(* IEC 61131-3 sources: plc_simulator/services/codesys/POUs (part 5) *)

(* ---- STC_SortTasks.st ---- *)
(* ===========================================================================================
 *  STC_SortTasks — Insertion sort task queues by priority
 *
 *  Company : Galvatek part of the John Cockerill Group
 *  Author  : Jarmo Piipponen
 *  Created : 25.03.2026
 *
 * -------------------------------------------------------------------------------------------
 *  Shared FC: both TSK and DEP call this with different arrays.
 *  Priority: emergency (overtime ratio > 1.0) first, then
 *  earliest StartTime.
 *
 *  ------------------------------------------------------------------------------------------
 *
 *  Changes:
 *
 *
 *
 *)

FUNCTION STC_SortTasks : BOOL

(* Introduction of Variables ----------------------------------------------------------------*)

VAR_INPUT
  i_trans                   : INT;    (* 0 = all, 1..3 = specific transporter *)
  i_time_s                  : LINT;
END_VAR

VAR_IN_OUT  (* array sizes must match GVL_JC_Constants: 3=MAX_TRANSPORTERS, 10=MAX_UNITS *)
  io_task                   : ARRAY[1..3] OF UDT_JC_TskQueueType;
  io_batch                  : ARRAY[1..10] OF UDT_BatchType;
END_VAR

VAR_EXTERNAL CONSTANT
    MAX_TRANSPORTERS        : INT;
    MAX_UNITS               : INT;
    IN_PROCESS              : INT;
END_VAR

VAR_EXTERNAL
  g_unit                    : ARRAY[1..MAX_UNITS] OF UDT_JC_UnitType;
END_VAR

VAR
  ti                        : INT;
  t_start                   : INT;
  t_end                     : INT;
  ins_i                     : INT;
  ins_j                     : INT;
  ins_cnt                   : INT;
  tmp_task                  : UDT_JC_TskTaskType;
  tmp_unit                  : INT;
  cur_unit                  : INT;
  tmp_ratio                 : REAL;
  cur_ratio                 : REAL;
  tmp_emerg                 : BOOL;
  cur_emerg                 : BOOL;
  do_shift                  : BOOL;
END_VAR

STC_SortTasks := TRUE;

IF i_trans >= 1 AND i_trans <= 3 THEN
  t_start := i_trans;
  t_end   := i_trans;
ELSE
  t_start := 1;
  t_end   := 3;
END_IF;

FOR ti := t_start TO t_end DO
  ins_cnt := io_task[ti].Count;
  IF ins_cnt >= 2 THEN
    FOR ins_i := 2 TO ins_cnt DO
      tmp_task := io_task[ti].Queue[ins_i];

      tmp_ratio := 0.0;
      tmp_unit  := tmp_task.Unit;
      IF tmp_unit >= 1 AND tmp_unit <= MAX_UNITS THEN
        IF io_batch[tmp_unit].State = IN_PROCESS
           AND tmp_task.Stage >= 1 THEN
          IF io_batch[tmp_unit].CurStage = tmp_task.Stage
             AND g_unit[tmp_unit].location = tmp_task.LiftStationTarget
             AND io_batch[tmp_unit].StartTime > LINT#0
             AND io_batch[tmp_unit].MaxTime > 0 THEN
            tmp_ratio := LINT_TO_REAL(i_time_s - io_batch[tmp_unit].StartTime)
                         / DINT_TO_REAL(io_batch[tmp_unit].MaxTime);
          END_IF;
        END_IF;
      END_IF;
      tmp_emerg := tmp_ratio > 1.0;

      ins_j := 0;
      FOR ins_j := ins_i - 1 TO 1 BY -1 DO
        cur_ratio := 0.0;
        cur_unit  := io_task[ti].Queue[ins_j].Unit;
        IF cur_unit >= 1 AND cur_unit <= MAX_UNITS THEN
          IF io_batch[cur_unit].State = IN_PROCESS
             AND io_task[ti].Queue[ins_j].Stage >= 1 THEN
            IF io_batch[cur_unit].CurStage = io_task[ti].Queue[ins_j].Stage
               AND g_unit[cur_unit].location = io_task[ti].Queue[ins_j].LiftStationTarget
               AND io_batch[cur_unit].StartTime > LINT#0
               AND io_batch[cur_unit].MaxTime > 0 THEN
              cur_ratio := LINT_TO_REAL(i_time_s - io_batch[cur_unit].StartTime)
                           / DINT_TO_REAL(io_batch[cur_unit].MaxTime);
            END_IF;
          END_IF;
        END_IF;
        cur_emerg := cur_ratio > 1.0;

        do_shift := FALSE;
        IF tmp_emerg AND NOT cur_emerg THEN
          do_shift := TRUE;
        ELSIF tmp_emerg AND cur_emerg THEN
          IF tmp_ratio > cur_ratio THEN
            do_shift := TRUE;
          END_IF;
        ELSIF NOT tmp_emerg AND NOT cur_emerg THEN
          IF io_task[ti].Queue[ins_j].StartTime > tmp_task.StartTime THEN
            do_shift := TRUE;
          END_IF;
        END_IF;

        IF NOT do_shift THEN EXIT; END_IF;

        io_task[ti].Queue[ins_j + 1] := io_task[ti].Queue[ins_j];
      END_FOR;

      io_task[ti].Queue[ins_j + 1] := tmp_task;
    END_FOR;
  END_IF;
END_FOR;

END_FUNCTION

(* ---- STC_SwapTasks.st ---- *)
(* ===========================================================================================
 *  STC_SwapTasks — Swap same-station task pairs
 *
 *  Company : Galvatek part of the John Cockerill Group
 *  Author  : Jarmo Piipponen
 *  Created : 25.03.2026
 *
 * -------------------------------------------------------------------------------------------
 *  Shared FC: both TSK and DEP call this with different arrays.
 *  Swaps adjacent tasks on the same transporter when the first
 *  task's sink equals the second task's lift (chain optimization).
 *  Returns swap count.
 *
 *  ------------------------------------------------------------------------------------------
 *
 *  Changes:
 *
 *
 *
 *)

FUNCTION STC_SwapTasks : INT   (* returns swap count *)

(* Introduction of Variables ----------------------------------------------------------------*)

VAR_IN_OUT  (* array sizes must match GVL_JC_Constants: 3=MAX_TRANSPORTERS *)
  io_task                   : ARRAY[1..3] OF UDT_JC_TskQueueType;
END_VAR

VAR_EXTERNAL CONSTANT
    MAX_TRANSPORTERS        : INT;
END_VAR

VAR
  ti                        : INT;
  qi                        : INT;
  cnt                       : INT;
  tmp                       : UDT_JC_TskTaskType;
  swaps                     : INT;
END_VAR

swaps := 0;

FOR ti := 1 TO MAX_TRANSPORTERS DO
  cnt := io_task[ti].Count;
  IF cnt >= 2 THEN
    FOR qi := 1 TO cnt - 1 DO
      IF io_task[ti].Queue[qi].Unit <> io_task[ti].Queue[qi + 1].Unit
         AND io_task[ti].Queue[qi].SinkStationTarget = io_task[ti].Queue[qi + 1].LiftStationTarget THEN
        tmp := io_task[ti].Queue[qi];
        io_task[ti].Queue[qi] := io_task[ti].Queue[qi + 1];
        io_task[ti].Queue[qi + 1] := tmp;
        swaps := swaps + 1;
      END_IF;
    END_FOR;
  END_IF;
END_FOR;

STC_SwapTasks := swaps;

END_FUNCTION

(* ---- STC_TakeOut.st ---- *)
(* STC_TakeOut - Evaluate and trigger idle take-out for transporters
   Uses station-specific TakeOutDelay (seconds) and TakeOutDistance (mm) *)
(* IMPORT_MARKER_2026_04_01_B *)

FUNCTION STC_TakeOut : BOOL

VAR_INPUT
  i_time_s                  : LINT;
END_VAR

VAR
  ti                        : INT;
  current_station           : INT;
  take_out_delay            : INT;
  take_out_dist             : DINT;
  idle_time                 : LINT;
  current_x                 : DINT;
  target_x                  : DINT;
  next_lift_x               : DINT;
  area_center               : DINT;
  dir                       : INT;
  queued_lift_station       : INT;
  time_to_start             : LINT;
  si                        : INT;
  stn_x                     : DINT;
  best_stn                  : INT;
  best_dist                 : DINT;
  dx                        : DINT;
END_VAR

STC_TakeOut := TRUE;

FOR ti := 1 TO MAX_TRANSPORTERS DO

  IF g_transporter[ti].Phase <> 0 THEN CONTINUE; END_IF;
  IF g_transporter[ti].Status <> 3 THEN CONTINUE; END_IF;
  IF NOT g_transporter[ti].IsActive THEN CONTINUE; END_IF;

  current_station := g_transporter[ti].CurrentStation;
  IF current_station < MIN_STATION_INDEX OR current_station > MAX_STATION_INDEX THEN CONTINUE; END_IF;

  take_out_delay := Stations[current_station].TakeOutDelay;
  IF take_out_delay = 0 THEN CONTINUE; END_IF;

  take_out_dist := INT_TO_DINT(Stations[current_station].TakeOutDistance);
  IF take_out_dist <= 0 THEN CONTINUE; END_IF;

  idle_time := i_time_s - g_transporter[ti].IdleStartTime;
  IF idle_time < DINT_TO_LINT(INT_TO_DINT(take_out_delay)) THEN CONTINUE; END_IF;

  (* Defer if next task on SAME station starts soon *)
  IF g_task[ti].Count > 0 THEN
    queued_lift_station := g_task[ti].Queue[1].LiftStationTarget;
    IF queued_lift_station = current_station THEN
      time_to_start := g_task[ti].Queue[1].StartTime - i_time_s;
      IF time_to_start >= 0 AND time_to_start < DINT_TO_LINT(INT_TO_DINT(TAKE_OUT_MIN_WAIT_S)) THEN
        CONTINUE;
      END_IF;
    END_IF;
  END_IF;

  current_x := g_transporter[ti].XPosition;

  (* Determine direction: toward next task or toward area center *)
  IF g_task[ti].Count > 0 THEN
    next_lift_x := Stations[g_task[ti].Queue[1].LiftStationTarget].XPosition;
    IF next_lift_x > current_x THEN
      dir := 1;
    ELSE
      dir := -1;
    END_IF;
  ELSE
    area_center := (Transporters[ti].DrivePosMin + Transporters[ti].DrivePosMax) / 2;
    IF area_center > current_x THEN
      dir := 1;
    ELSE
      dir := -1;
    END_IF;
  END_IF;

  (* Compute minimum target position from TakeOutDistance *)
  target_x := current_x + (INT_TO_DINT(dir) * take_out_dist);

  (* Find nearest station in move direction that is at least take_out_dist away *)
  best_stn := 0;
  best_dist := DINT#2147483647;
  FOR si := MIN_STATION_INDEX TO MIN_STATION_INDEX + CountStations - 1 DO
    stn_x := Stations[si].XPosition;
    IF stn_x = 0 THEN CONTINUE; END_IF;
    (* Station must be in the correct direction and at least take_out_dist from current *)
    IF dir > 0 THEN
      dx := stn_x - current_x;
    ELSE
      dx := current_x - stn_x;
    END_IF;
    IF dx >= take_out_dist AND dx < best_dist THEN
      (* Must be within transporter drive limits *)
      IF stn_x >= Transporters[ti].DrivePosMin AND stn_x <= Transporters[ti].DrivePosMax THEN
        best_dist := dx;
        best_stn := si;
      END_IF;
    END_IF;
  END_FOR;

  IF best_stn > 0 THEN
    target_x := Stations[best_stn].XPosition;
  ELSE
    CONTINUE;  (* no station found in direction — skip take-out *)
  END_IF;

  (* Skip if we can't actually move *)
  IF ABS(target_x - current_x) < 100 THEN CONTINUE; END_IF;

  (* If next task starts soon and take-out would pass over its lift station,
     stop at the lift station instead *)
  IF g_task[ti].Count > 0 THEN
    time_to_start := g_task[ti].Queue[1].StartTime - i_time_s;
    IF time_to_start >= 0 AND time_to_start < DINT_TO_LINT(INT_TO_DINT(TAKE_OUT_MIN_WAIT_S)) THEN
      queued_lift_station := g_task[ti].Queue[1].LiftStationTarget;
      IF queued_lift_station >= MIN_STATION_INDEX AND queued_lift_station <= MAX_STATION_INDEX THEN
        next_lift_x := Stations[queued_lift_station].XPosition;
        (* Check if take-out target is on the other side of lift station *)
        IF dir > 0 AND target_x > next_lift_x AND next_lift_x > current_x THEN
          target_x := next_lift_x;
        ELSIF dir < 0 AND target_x < next_lift_x AND next_lift_x < current_x THEN
          target_x := next_lift_x;
        END_IF;
      END_IF;
    END_IF;
  END_IF;

  (* Re-check: still worth moving? *)
  IF ABS(target_x - current_x) < 100 THEN CONTINUE; END_IF;

  g_transporter[ti].Phase := 1;
  g_transporter[ti].LiftStationTarget := 0;
  g_transporter[ti].SinkStationTarget := 0;
  g_transporter[ti].XDriveTarget := target_x;
  g_transporter[ti].XFinalTarget := target_x;

END_FOR;

STC_TakeOut := TRUE;

END_FUNCTION

(* ---- STC_TrackMoveTimes.st ---- *)
(* ===========================================================================================
 *  STC_TrackMoveTimes — Record phase transition timestamps
 *
 *  Company : Galvatek part of the John Cockerill Group
 *  Author  : Jarmo Piipponen
 *  Created : 25.03.2026
 *
 * -------------------------------------------------------------------------------------------
 *  Called from SIM code at each transporter phase change.
 *  Uses g_time_100ms (0.1s ticks). On 4→0 completion,
 *  calculates net durations and updates g_move[] with
 *  weighted average: new = (old * 4 + measured) / 5.
 *
 *  ------------------------------------------------------------------------------------------
 *
 *  Changes:
 *
 *
 *
 *)

FUNCTION STC_TrackMoveTimes : BOOL

(* Introduction of Variables ----------------------------------------------------------------*)

VAR_INPUT
  i_trans                   : INT;   (* transporter index 1..MAX_TRANSPORTERS *)
  i_prev                    : INT;   (* previous phase *)
  i_new                     : INT;   (* new phase *)
END_VAR

VAR_EXTERNAL CONSTANT
    MAX_TRANSPORTERS        : INT;
    MIN_STATION_INDEX        : INT;
    MAX_STATION_INDEX        : INT;
END_VAR

VAR_EXTERNAL
  g_transporter             : ARRAY[1..MAX_TRANSPORTERS] OF UDT_TransporterStatusType;
  Stations                 : ARRAY[MIN_STATION_INDEX..MAX_STATION_INDEX] OF UDT_StationType;
  Transporters                     : ARRAY[0..MAX_TRANSPORTERS] OF UDT_TransporterType;
  g_move                    : ARRAY[1..MAX_TRANSPORTERS] OF UDT_JC_MoveTimesType;
  g_actual_move             : ARRAY[1..MAX_TRANSPORTERS] OF UDT_JC_ActualMoveTimeType;
  g_time_s                  : LINT;
  g_time_100ms              : LINT;
END_VAR

VAR
  t                         : INT;
  lift_stn                  : INT;
  sink_stn                  : INT;
  start_stn                 : INT;
  li                        : INT;   (* lift station index = stn - 100 *)
  si                        : INT;   (* sink station index = stn - 100 *)
  st_i                      : INT;   (* start station index = stn - 100 *)
  raw_lift                  : INT;   (* measured lift duration in 0.1s ticks *)
  raw_sink                  : INT;   (* measured sink duration in 0.1s ticks *)
  raw_trav1                 : INT;   (* measured travel start→lift in 0.1s ticks *)
  raw_trav2                 : INT;   (* measured travel lift→sink in 0.1s ticks *)
  drip_x10                  : INT;   (* DrippingTime in 0.1s ticks from lift station *)
  tray_x10                  : INT;   (* DripTrayDelay in 0.1s ticks from transporter config *)
  dev_x10                   : INT;   (* DeviceDelay in 0.1s ticks from sink station *)
END_VAR

t := i_trans;

(* Bounds check *)
IF t < 1 OR t > MAX_TRANSPORTERS THEN
    RETURN;
END_IF;

CASE i_prev OF
    0: (* 0→1 : siirto nostoasemalle alkaa *)
        IF i_new = 1 THEN
            g_actual_move[t].StartStation := g_transporter[t].CurrentStation;
            g_actual_move[t].LiftStation  := g_transporter[t].LiftStationTarget;
            g_actual_move[t].SinkStation  := g_transporter[t].SinkStationTarget;
            g_actual_move[t].ts0 := g_time_100ms;
            g_actual_move[t].Invalidated := FALSE;
        END_IF;
    1: (* 1→2 : nosto alkaa *)
        IF i_new = 2 THEN
            g_actual_move[t].ts1 := g_time_100ms;
        END_IF;
    2: (* 2→3 : siirto laskuasemalle alkaa *)
        IF i_new = 3 THEN
            g_actual_move[t].ts2 := g_time_100ms;
        END_IF;
    3: (* 3→4 : lasku alkaa *)
        IF i_new = 4 THEN
            g_actual_move[t].ts3 := g_time_100ms;
        END_IF;
    4: (* 4→0 : handled after CASE — see below *)
END_CASE;

(* ── Invalidate on anomaly (checked at every phase transition) ── *)
IF i_new > 0 THEN
    (* Not in automatic mode: task interrupted *)
    IF g_transporter[t].Status < 4 THEN
        g_actual_move[t].Invalidated := TRUE;
    END_IF;
    (* Transporter fault active *)
    IF g_transporter[t].Fault THEN
        g_actual_move[t].Invalidated := TRUE;
    END_IF;
END_IF;

(* ── 4→0 completion: calculate and update g_move ── *)
IF i_prev = 4 AND i_new = 0 THEN
    g_actual_move[t].ts4 := g_time_100ms;

    (* Only update if all timestamps are valid and transfer was normal *)
    IF g_actual_move[t].ts0 > 0
       AND g_actual_move[t].ts1 > 0
       AND g_actual_move[t].ts2 > 0
       AND g_actual_move[t].ts3 > 0
       AND NOT g_actual_move[t].Invalidated
    THEN
                lift_stn  := g_actual_move[t].LiftStation;
                sink_stn  := g_actual_move[t].SinkStation;
                start_stn := g_actual_move[t].StartStation;
                li   := lift_stn  - MIN_STATION_INDEX;
                si   := sink_stn  - MIN_STATION_INDEX;
                st_i := start_stn - MIN_STATION_INDEX;

                (* Mechanical delays in 0.1s ticks *)
                drip_x10 := Stations[lift_stn].DrippingTime;
                tray_x10 := Transporters[t].DripTrayDelay;
                dev_x10  := Stations[sink_stn].DeviceDelay;

                (* Raw durations are already in 0.1s ticks *)
                raw_trav1 := LINT_TO_INT(g_actual_move[t].ts1 - g_actual_move[t].ts0);
                raw_trav2 := LINT_TO_INT(g_actual_move[t].ts3 - g_actual_move[t].ts2);

                (* Net lift = (ts2-ts1) - DrippingTime - DripTrayDelay *)
                raw_lift := LINT_TO_INT(g_actual_move[t].ts2 - g_actual_move[t].ts1)
                            - drip_x10 - tray_x10;

                (* Net sink = (ts4-ts3) - DripTrayDelay - DeviceDelay *)
                raw_sink := LINT_TO_INT(g_actual_move[t].ts4 - g_actual_move[t].ts3)
                            - tray_x10 - dev_x10;

                (* Clamp to minimum 0 *)
  IF raw_lift < 0 THEN raw_lift := 0; END_IF;
  IF raw_sink < 0 THEN raw_sink := 0; END_IF;
  IF raw_trav1 < 0 THEN raw_trav1 := 0; END_IF;
  IF raw_trav2 < 0 THEN raw_trav2 := 0; END_IF;

                (* Bounds check indices *)
                IF li >= 1 AND li <= 30
                   AND si >= 1 AND si <= 30
                   AND st_i >= 1 AND st_i <= 30
                THEN
                    (* Weighted average: new = (old * 4 + measured) / 5 *)

                    (* Lift time at lift station *)
                    g_move[t].LiftTime[li] :=
                        (g_move[t].LiftTime[li] * 4 + raw_lift) / 5;

                    (* Sink time at sink station *)
                    g_move[t].SinkTime[si] :=
                        (g_move[t].SinkTime[si] * 4 + raw_sink) / 5;

                    (* Travel: lift → sink (both directions) — phase 3 is always exact station-to-station *)
                    g_move[t].Travel[li].ToTime[si] :=
                        (g_move[t].Travel[li].ToTime[si] * 4 + raw_trav2) / 5;
                    g_move[t].Travel[si].ToTime[li] :=
                        (g_move[t].Travel[si].ToTime[li] * 4 + raw_trav2) / 5;
                END_IF;
            END_IF;
END_IF;

STC_TrackMoveTimes := TRUE;

END_FUNCTION

(* ---- STC_UpdateUnitLocation.st ---- *)
(* ===========================================================================================
 *  STC_UpdateUnitLocation — Update a unit's location
 *
 *  Company : Galvatek part of the John Cockerill Group
 *  Author  : Jarmo Piipponen
 *  Created : 25.03.2026
 *
 * -------------------------------------------------------------------------------------------
 *  Sets g_unit[i_unit].location to the given new location.
 *  Updates g_station_occupancy[].UnitId + ChangeTime for both old
 *  and new locations.
 *
 *  When moving to a station:
 *  - Advances batch CurStage if batch is IN_PROCESS
 *  - Updates batch min/max/cal times from treatment program
 *  - Clears unit target if i_ntt_primary = 1
 *
 *  ------------------------------------------------------------------------------------------
 *
 *  Changes:
 *
 *
 *
 *)

FUNCTION STC_UpdateUnitLocation : BOOL

(* Introduction of Variables ----------------------------------------------------------------*)

VAR_INPUT
  i_unit                    : INT;   (* unit number to update *)
  i_location                : INT;   (* new location: <100 = transporter id, >=100 = station number *)
  i_ntt_primary             : INT;   (* 1 = sink is NTT primary → clear target, 0 = don't clear *)
END_VAR

VAR_EXTERNAL CONSTANT
    MAX_UNITS               : INT;
    MAX_TRANSPORTERS        : INT;
    MAX_STEPS_PER_PROGRAM   : INT;
    MIN_STATION_INDEX        : INT;
    MAX_STATION_INDEX        : INT;
    IN_PROCESS              : INT;
    USED                    : INT;
    TO_NONE                 : INT;
END_VAR

VAR_EXTERNAL
  g_unit                    : ARRAY[1..MAX_UNITS] OF UDT_JC_UnitType;
  Stations                 : ARRAY[MIN_STATION_INDEX..MAX_STATION_INDEX] OF UDT_StationType;
  g_station_occupancy             : ARRAY[1..MAX_STATION_INDEX] OF UDT_JC_UnitAtStationType;
  g_batch                   : ARRAY[1..MAX_UNITS] OF UDT_BatchType;
  TreatmentPrograms                 : ARRAY[1..MAX_UNITS] OF UDT_TreatmentProgramType;
  g_transporter             : ARRAY[1..MAX_TRANSPORTERS] OF UDT_TransporterStatusType;
  g_move                    : ARRAY[1..MAX_TRANSPORTERS] OF UDT_JC_MoveTimesType;
  g_time_s                  : LINT;
END_VAR

VAR
  old_loc                   : INT;
  new_stg                   : INT;
END_VAR

IF (i_unit >= 1) AND (i_unit <= MAX_UNITS) THEN
  old_loc := g_unit[i_unit].location;

  (* --- Clear unit_id from old location (unified: transporter or station) --- *)
  IF (old_loc >= 1) AND (old_loc <= MAX_STATION_INDEX) THEN
    g_station_occupancy[old_loc].UnitId     := 0;
    g_station_occupancy[old_loc].ChangeTime := g_time_s;
  END_IF;

  (* --- Update unit location --- *)
  g_unit[i_unit].location := i_location;

  (* --- Set unit_id on new location (unified: transporter or station) --- *)
  IF (i_location >= 1) AND (i_location <= MAX_STATION_INDEX) THEN
    g_station_occupancy[i_location].UnitId     := i_unit;
    g_station_occupancy[i_location].ChangeTime := g_time_s;

    (* Station-specific: batch stage advance only when landing on a station *)
    IF (i_location >= MIN_STATION_INDEX) THEN

    (* Advance batch stage if unit is USED with an active batch *)
    IF (g_unit[i_unit].Status = USED)  (* USED *)
       AND (g_batch[i_unit].BatchCode <> 0)
       AND (g_batch[i_unit].State = IN_PROCESS)
       AND (g_batch[i_unit].CurStage < MAX_STEPS_PER_PROGRAM) THEN
      g_batch[i_unit].CurStage := g_batch[i_unit].CurStage + 1;

      (* Stamp arrival time on new station — used by CalcSchedule for elapsed calculation *)
      g_batch[i_unit].StartTime := g_time_s;

      (* Update batch treatment times from program for the new stage *)
      IF (TreatmentPrograms[i_unit].ProgramId = g_batch[i_unit].ProgId)
         AND (TreatmentPrograms[i_unit].ProgramId > 0) THEN
        new_stg := g_batch[i_unit].CurStage;
        IF (new_stg >= 1) AND (new_stg <= MAX_STEPS_PER_PROGRAM) THEN
          g_batch[i_unit].MinTime := TreatmentPrograms[i_unit].Steps[new_stg].MinTime;
          g_batch[i_unit].MaxTime := TreatmentPrograms[i_unit].Steps[new_stg].MaxTime;
          g_batch[i_unit].CalTime := TreatmentPrograms[i_unit].Steps[new_stg].CalTime;
        END_IF;
      END_IF;
    END_IF;

    (* NOT_PROCESSED batch on station: clear times so UI shows no progress bar *)
    IF (g_batch[i_unit].BatchCode <> 0)
       AND (g_batch[i_unit].State <> IN_PROCESS) THEN
      g_batch[i_unit].MinTime   := 0;
      g_batch[i_unit].CalTime   := 0;
      g_batch[i_unit].MaxTime   := 32000;  (* ~8.9 h cap, INT max safe *)
      g_batch[i_unit].StartTime := g_time_s;
    END_IF;

    (* Clear unit target ONLY when i_ntt_primary = 1 (primary NTT destination).
       All other cases: keep target so NTT retries primary later. *)
    IF g_unit[i_unit].Target <> TO_NONE AND i_ntt_primary > 0 THEN
      g_unit[i_unit].Target := TO_NONE;  (* primary reached → clear *)
    END_IF;

    END_IF; (* i_location >= MIN_STATION_INDEX — station-specific block *)
  END_IF; (* i_location valid *)
END_IF;

STC_UpdateUnitLocation := TRUE;

END_FUNCTION

(* ---- TSK_Analyze.st ---- *)
(* ===========================================================================================
 *  TSK_Analyze — Conflict analysis for task list
 *
 *  Company : Galvatek part of the John Cockerill Group
 *  Author  : Jarmo Piipponen
 *  Created : 25.03.2026
 *
 * -------------------------------------------------------------------------------------------
 *  Read-only analysis: never writes globals.
 *
 *  Three conflict checks, each stops at first hit:
 *  1. TASK_SEQUENCE
 *  2. CROSS_TRANSPORTER_HANDOFF
 *  3. TRANSPORTER_COLLISION
 *
 *  ------------------------------------------------------------------------------------------
 *
 *  Changes:
 *
 *
 *
 *)

FUNCTION TSK_Analyze : BOOL

(* Introduction of Variables ----------------------------------------------------------------*)

VAR_IN_OUT  (* array sizes must match GVL_JC_Constants: 3=MAX_TRANSPORTERS *)
  io_task                   : ARRAY[1..3] OF UDT_JC_TskQueueType;
END_VAR

VAR_EXTERNAL CONSTANT
    MAX_TRANSPORTERS        : INT;
    MAX_UNITS               : INT;
    MIN_STATION_INDEX        : INT;
    MAX_STATION_INDEX        : INT;
END_VAR

VAR_EXTERNAL
  Stations                 : ARRAY[MIN_STATION_INDEX..MAX_STATION_INDEX] OF UDT_StationType;
  g_move                    : ARRAY[1..MAX_TRANSPORTERS] OF UDT_JC_MoveTimesType;
END_VAR

VAR_OUTPUT
  o_has_conflict            : BOOL;
  o_conf_type               : INT;     (* 1=TASK_SEQUENCE, 2=COLLISION, 3=HANDOFF *)
  o_conf_unit               : INT;
  o_conf_stage              : INT;
  o_conf_trans              : INT;
  o_blocked_unit            : INT;
  o_blocked_stage           : INT;
  o_deficit                 : REAL;
  checked_count             : INT;
END_VAR

VAR
  ti                        : INT;
  tj                        : INT;
  qi                        : INT;
  qj                        : INT;
  prev_sink                 : INT;
  next_lift                 : INT;
  travel_s                  : REAL;
  gap_s                     : REAL;
  deficit_s                 : REAL;
  lift_x                    : REAL;
  sink_x                    : REAL;
  x1_min                    : REAL;
  x1_max                    : REAL;
  x2_min                    : REAL;
  x2_max                    : REAL;
  xo_start                  : REAL;
  xo_end                    : REAL;
  to_start                  : LINT;
  to_end                    : LINT;
  l_idx                     : INT;
  s_idx                     : INT;
  lift_x2                   : REAL;
  sink_x2                   : REAL;
  l_idx2                    : INT;
  s_idx2                    : INT;
  cur_unit                  : INT;
  cur_stage                 : INT;
  found_next                : BOOL;
  recv_prev_end             : LINT;
  recv_prev_sink            : INT;
  has_recv_prev             : BOOL;
  rk                        : INT;
  recv_prev_unit            : INT;
  recv_prev_stg             : INT;
  recv_travel               : REAL;
  recv_earliest             : LINT;
  handoff_deficit           : REAL;
  total_tasks               : INT;
  DEFICIT_TOL               : REAL := 1.0;
  tmp_move                  : UDT_JC_MoveTimesType;
END_VAR

TSK_Analyze := FALSE;
o_has_conflict := FALSE;
o_conf_type    := 0;
o_deficit      := 0.0;
checked_count  := 0;

total_tasks := 0;
FOR ti := 1 TO MAX_TRANSPORTERS DO
  total_tasks := total_tasks + io_task[ti].Count;
END_FOR;
IF total_tasks = 0 THEN RETURN; END_IF;

(* CHECK 1: TASK_SEQUENCE *)
FOR ti := 1 TO MAX_TRANSPORTERS DO
  FOR qi := 1 TO io_task[ti].Count - 1 DO
    IF io_task[ti].Queue[qi].Unit > 0 AND io_task[ti].Queue[qi + 1].Unit > 0 THEN
      prev_sink := io_task[ti].Queue[qi].SinkStationTarget;
      next_lift := io_task[ti].Queue[qi + 1].LiftStationTarget;
      tmp_move := g_move[ti];
      travel_s := STC_CalcHorizontalTravel(i_from_stn := prev_sink, i_to_stn := next_lift, i_move := tmp_move);
      gap_s := LINT_TO_REAL(io_task[ti].Queue[qi + 1].StartTime - io_task[ti].Queue[qi].FinishTime);
      deficit_s := travel_s - gap_s;
      IF deficit_s > DEFICIT_TOL THEN
  o_has_conflict := TRUE;
  o_conf_type := 1;
        o_conf_unit := io_task[ti].Queue[qi + 1].Unit;
        o_conf_stage := io_task[ti].Queue[qi + 1].Stage;
        o_conf_trans := ti;
        o_blocked_unit := io_task[ti].Queue[qi].Unit;
        o_blocked_stage := io_task[ti].Queue[qi].Stage;
  o_deficit := deficit_s;
  checked_count := total_tasks;
  TSK_Analyze := TRUE; RETURN;
      END_IF;
    END_IF;
  END_FOR;
END_FOR;

(* CHECK 2: CROSS_TRANSPORTER_HANDOFF *)
FOR ti := 1 TO MAX_TRANSPORTERS DO
  FOR qi := 1 TO io_task[ti].Count DO
    cur_unit  := io_task[ti].Queue[qi].Unit;
    cur_stage := io_task[ti].Queue[qi].Stage;
    IF cur_unit > 0 THEN
      found_next := FALSE;
      FOR tj := 1 TO MAX_TRANSPORTERS DO
        IF tj <> ti AND NOT found_next THEN
          FOR qj := 1 TO io_task[tj].Count DO
            IF NOT found_next THEN
              IF io_task[tj].Queue[qj].Unit = cur_unit
                 AND io_task[tj].Queue[qj].Stage = cur_stage + 1 THEN
                found_next := TRUE;
                has_recv_prev := FALSE;
  recv_prev_end := 0;
  recv_prev_sink := 0;
  recv_prev_unit := 0;
  recv_prev_stg := 0;
                FOR rk := 1 TO io_task[tj].Count DO
                  IF rk <> qj THEN
                    IF io_task[tj].Queue[rk].FinishTime <= io_task[tj].Queue[qj].StartTime THEN
                      IF NOT has_recv_prev OR io_task[tj].Queue[rk].FinishTime > recv_prev_end THEN
                        has_recv_prev := TRUE;
                        recv_prev_end  := io_task[tj].Queue[rk].FinishTime;
                        recv_prev_sink := io_task[tj].Queue[rk].SinkStationTarget;
                        recv_prev_unit := io_task[tj].Queue[rk].Unit;
                        recv_prev_stg  := io_task[tj].Queue[rk].Stage;
                      END_IF;
                    END_IF;
                  END_IF;
                END_FOR;
                IF has_recv_prev THEN
                  recv_travel := STC_CalcHorizontalTravel(
                    i_from_stn := recv_prev_sink,
                    i_to_stn   := io_task[ti].Queue[qi].SinkStationTarget,
                    i_move     := g_move[tj]);
                  recv_earliest := recv_prev_end + REAL_TO_LINT(recv_travel);
                  handoff_deficit := LINT_TO_REAL(recv_earliest - io_task[ti].Queue[qi].FinishTime);
                  IF handoff_deficit > DEFICIT_TOL THEN
  o_has_conflict := TRUE;
  o_conf_type := 3;
                    o_conf_unit := io_task[ti].Queue[qi].Unit;
                    o_conf_stage := io_task[ti].Queue[qi].Stage;
                    o_conf_trans := ti;
                    o_blocked_unit := recv_prev_unit;
                    o_blocked_stage := recv_prev_stg;
  o_deficit := handoff_deficit;
  checked_count := total_tasks;
  TSK_Analyze := TRUE; RETURN;
                  END_IF;
                END_IF;
              END_IF;
            END_IF;
          END_FOR;
        END_IF;
      END_FOR;
    END_IF;
  END_FOR;
END_FOR;

(* CHECK 3: TRANSPORTER_COLLISION *)
FOR ti := 1 TO MAX_TRANSPORTERS DO
  FOR qi := 1 TO io_task[ti].Count DO
    IF io_task[ti].Queue[qi].Unit > 0 THEN
      l_idx := io_task[ti].Queue[qi].LiftStationTarget - MIN_STATION_INDEX;
      s_idx := io_task[ti].Queue[qi].SinkStationTarget - MIN_STATION_INDEX;
      IF l_idx >= 1 AND l_idx <= 30 THEN
        lift_x := DINT_TO_REAL(Stations[io_task[ti].Queue[qi].LiftStationTarget].XPosition);
  ELSE lift_x := 0.0; END_IF;
      IF s_idx >= 1 AND s_idx <= 30 THEN
        sink_x := DINT_TO_REAL(Stations[io_task[ti].Queue[qi].SinkStationTarget].XPosition);
  ELSE sink_x := 0.0; END_IF;
  IF lift_x < sink_x THEN x1_min := lift_x;
  x1_max := sink_x;
  ELSE x1_min := sink_x;
  x1_max := lift_x; END_IF;

      FOR tj := ti + 1 TO MAX_TRANSPORTERS DO
        FOR qj := 1 TO io_task[tj].Count DO
          IF io_task[tj].Queue[qj].Unit > 0 THEN
            l_idx2 := io_task[tj].Queue[qj].LiftStationTarget - MIN_STATION_INDEX;
            s_idx2 := io_task[tj].Queue[qj].SinkStationTarget - MIN_STATION_INDEX;
            IF l_idx2 >= 1 AND l_idx2 <= 30 THEN
              lift_x2 := DINT_TO_REAL(Stations[io_task[tj].Queue[qj].LiftStationTarget].XPosition);
  ELSE lift_x2 := 0.0; END_IF;
            IF s_idx2 >= 1 AND s_idx2 <= 30 THEN
              sink_x2 := DINT_TO_REAL(Stations[io_task[tj].Queue[qj].SinkStationTarget].XPosition);
  ELSE sink_x2 := 0.0; END_IF;
  IF lift_x2 < sink_x2 THEN x2_min := lift_x2;
  x2_max := sink_x2;
  ELSE x2_min := sink_x2;
  x2_max := lift_x2; END_IF;

  xo_start := x1_min; IF x2_min > xo_start THEN xo_start := x2_min; END_IF;
  xo_end := x1_max; IF x2_max < xo_end THEN xo_end := x2_max; END_IF;

            IF xo_start < xo_end THEN
              to_start := io_task[ti].Queue[qi].StartTime;
  IF io_task[tj].Queue[qj].StartTime > to_start THEN to_start := io_task[tj].Queue[qj].StartTime; END_IF;
              to_end := io_task[ti].Queue[qi].FinishTime;
  IF io_task[tj].Queue[qj].FinishTime < to_end THEN to_end := io_task[tj].Queue[qj].FinishTime; END_IF;

              IF to_start < to_end THEN
                deficit_s := LINT_TO_REAL(to_end - to_start) + 2.0;
  o_has_conflict := TRUE;
  o_conf_type := 2;
                IF io_task[ti].Queue[qi].StartTime <= io_task[tj].Queue[qj].StartTime THEN
                  o_conf_unit := io_task[tj].Queue[qj].Unit;
                  o_conf_stage := io_task[tj].Queue[qj].Stage;
                  o_conf_trans := tj;
                  o_blocked_unit := io_task[ti].Queue[qi].Unit;
                  o_blocked_stage := io_task[ti].Queue[qi].Stage;
                ELSE
                  o_conf_unit := io_task[ti].Queue[qi].Unit;
                  o_conf_stage := io_task[ti].Queue[qi].Stage;
                  o_conf_trans := ti;
                  o_blocked_unit := io_task[tj].Queue[qj].Unit;
                  o_blocked_stage := io_task[tj].Queue[qj].Stage;
                END_IF;
  o_deficit := deficit_s;
  checked_count := total_tasks;
  TSK_Analyze := TRUE; RETURN;
              END_IF;
            END_IF;
          END_IF;
        END_FOR;
      END_FOR;
    END_IF;
  END_FOR;
END_FOR;

checked_count := total_tasks;

END_FUNCTION

(* ---- TSK_FC_Analyze.st ---- *)
(* ===========================================================================================
 *  TSK_FC_Analyze — Conflict analysis for task list
 *
 *  Company : Galvatek part of the John Cockerill Group
 *  Author  : Jarmo Piipponen
 *  Created : 25.03.2026
 *
 * -------------------------------------------------------------------------------------------
 *  Read-only analysis: never writes globals.
 *
 *  Three conflict checks, each stops at first hit:
 *  1. TASK_SEQUENCE
 *  2. CROSS_TRANSPORTER_HANDOFF
 *  3. TRANSPORTER_COLLISION
 *
 *  ------------------------------------------------------------------------------------------
 *
 *  Changes:
 *
 *
 *
 *)

FUNCTION TSK_FC_Analyze : BOOL

(* Introduction of Variables ----------------------------------------------------------------*)

VAR_IN_OUT  (* array sizes must match GVL_JC_Constants: 3=MAX_TRANSPORTERS *)
  ioTask                   : ARRAY[1..3] OF UDT_JC_TskQueueType;
END_VAR

VAR_EXTERNAL CONSTANT
    MAX_TRANSPORTERS        : INT;
    MAX_UNITS               : INT;
    MIN_STATION_INDEX        : INT;
    MAX_STATION_INDEX        : INT;
END_VAR

VAR_EXTERNAL
  Stations                 : ARRAY[MIN_STATION_INDEX..MAX_STATION_INDEX] OF UDT_StationType;
  Move                    : ARRAY[1..MAX_TRANSPORTERS] OF UDT_JC_MoveTimesType;
END_VAR

VAR_OUTPUT
  oHasConflict            : BOOL;
  oConfType               : INT;     (* 1=TASK_SEQUENCE, 2=COLLISION, 3=HANDOFF *)
  oConfUnit               : INT;
  oConfStage              : INT;
  oConfTrans              : INT;
  oBlockedUnit            : INT;
  oBlockedStage           : INT;
  oDeficit                 : REAL;
  oCheckedCount             : INT;
END_VAR

VAR
  vTi                        : INT;
  vTj                        : INT;
  vQi                        : INT;
  vQj                        : INT;
  vPrevSink                 : INT;
  vNextLift                 : INT;
  vTravelS                  : REAL;
  vGapS                     : REAL;
  vDeficitS                 : REAL;
  vLiftX                    : REAL;
  vSinkX                    : REAL;
  vX1Min                    : REAL;
  vX1Max                    : REAL;
  vX2Min                    : REAL;
  vX2Max                    : REAL;
  vXoStart                  : REAL;
  vXoEnd                    : REAL;
  vToStart                  : LINT;
  vToEnd                    : LINT;
  vLIdx                     : INT;
  vSIdx                     : INT;
  vLiftX2                   : REAL;
  vSinkX2                   : REAL;
  vLIdx2                    : INT;
  vSIdx2                    : INT;
  vCurUnit                  : INT;
  vCurStage                 : INT;
  vFoundNext                : BOOL;
  vRecvPrevEnd             : LINT;
  vRecvPrevSink            : INT;
  vHasRecvPrev             : BOOL;
  vRk                        : INT;
  vRecvPrevUnit            : INT;
  vRecvPrevStg             : INT;
  vRecvTravel               : REAL;
  vRecvEarliest             : LINT;
  vHandoffDeficit           : REAL;
  vTotalTasks               : INT;
  vDeficitTol               : REAL := 1.0;
  vTmpMove                  : UDT_JC_MoveTimesType;
END_VAR

TSK_FC_Analyze := FALSE;
oHasConflict := FALSE;
oConfType    := 0;
oDeficit      := 0.0;
oCheckedCount  := 0;

vTotalTasks := 0;
FOR vTi := 1 TO MAX_TRANSPORTERS DO
  vTotalTasks := vTotalTasks + ioTask[vTi].Count;
END_FOR;
IF vTotalTasks = 0 THEN RETURN; END_IF;

(* CHECK 1: TASK_SEQUENCE *)
FOR vTi := 1 TO MAX_TRANSPORTERS DO
  FOR vQi := 1 TO ioTask[vTi].Count - 1 DO
    IF ioTask[vTi].Queue[vQi].Unit > 0 AND ioTask[vTi].Queue[vQi + 1].Unit > 0 THEN
      vPrevSink := ioTask[vTi].Queue[vQi].SinkStationTarget;
      vNextLift := ioTask[vTi].Queue[vQi + 1].LiftStationTarget;
      vTmpMove := Move[vTi];
      vTravelS := STC_FC_CalcHorizontalTravel(iFromStn := vPrevSink, iToStn := vNextLift, iMove := vTmpMove);
      vGapS := LINT_TO_REAL(ioTask[vTi].Queue[vQi + 1].StartTime - ioTask[vTi].Queue[vQi].FinishTime);
      vDeficitS := vTravelS - vGapS;
      IF vDeficitS > vDeficitTol THEN
  oHasConflict := TRUE;
  oConfType := 1;
        oConfUnit := ioTask[vTi].Queue[vQi + 1].Unit;
        oConfStage := ioTask[vTi].Queue[vQi + 1].Stage;
        oConfTrans := vTi;
        oBlockedUnit := ioTask[vTi].Queue[vQi].Unit;
        oBlockedStage := ioTask[vTi].Queue[vQi].Stage;
  oDeficit := vDeficitS;
  oCheckedCount := vTotalTasks;
  TSK_FC_Analyze := TRUE; RETURN;
      END_IF;
    END_IF;
  END_FOR;
END_FOR;

(* CHECK 2: CROSS_TRANSPORTER_HANDOFF *)
FOR vTi := 1 TO MAX_TRANSPORTERS DO
  FOR vQi := 1 TO ioTask[vTi].Count DO
    vCurUnit  := ioTask[vTi].Queue[vQi].Unit;
    vCurStage := ioTask[vTi].Queue[vQi].Stage;
    IF vCurUnit > 0 THEN
      vFoundNext := FALSE;
      FOR vTj := 1 TO MAX_TRANSPORTERS DO
        IF vTj <> vTi AND NOT vFoundNext THEN
          FOR vQj := 1 TO ioTask[vTj].Count DO
            IF NOT vFoundNext THEN
              IF ioTask[vTj].Queue[vQj].Unit = vCurUnit
                 AND ioTask[vTj].Queue[vQj].Stage = vCurStage + 1 THEN
                vFoundNext := TRUE;
                vHasRecvPrev := FALSE;
  vRecvPrevEnd := 0;
  vRecvPrevSink := 0;
  vRecvPrevUnit := 0;
  vRecvPrevStg := 0;
                FOR vRk := 1 TO ioTask[vTj].Count DO
                  IF vRk <> vQj THEN
                    IF ioTask[vTj].Queue[vRk].FinishTime <= ioTask[vTj].Queue[vQj].StartTime THEN
                      IF NOT vHasRecvPrev OR ioTask[vTj].Queue[vRk].FinishTime > vRecvPrevEnd THEN
                        vHasRecvPrev := TRUE;
                        vRecvPrevEnd  := ioTask[vTj].Queue[vRk].FinishTime;
                        vRecvPrevSink := ioTask[vTj].Queue[vRk].SinkStationTarget;
                        vRecvPrevUnit := ioTask[vTj].Queue[vRk].Unit;
                        vRecvPrevStg  := ioTask[vTj].Queue[vRk].Stage;
                      END_IF;
                    END_IF;
                  END_IF;
                END_FOR;
                IF vHasRecvPrev THEN
                  vRecvTravel := STC_FC_CalcHorizontalTravel(
                    iFromStn := vRecvPrevSink,
                    iToStn   := ioTask[vTi].Queue[vQi].SinkStationTarget,
                    iMove     := Move[vTj]);
                  vRecvEarliest := vRecvPrevEnd + REAL_TO_LINT(vRecvTravel);
                  vHandoffDeficit := LINT_TO_REAL(vRecvEarliest - ioTask[vTi].Queue[vQi].FinishTime);
                  IF vHandoffDeficit > vDeficitTol THEN
  oHasConflict := TRUE;
  oConfType := 3;
                    oConfUnit := ioTask[vTi].Queue[vQi].Unit;
                    oConfStage := ioTask[vTi].Queue[vQi].Stage;
                    oConfTrans := vTi;
                    oBlockedUnit := vRecvPrevUnit;
                    oBlockedStage := vRecvPrevStg;
  oDeficit := vHandoffDeficit;
  oCheckedCount := vTotalTasks;
  TSK_FC_Analyze := TRUE; RETURN;
                  END_IF;
                END_IF;
              END_IF;
            END_IF;
          END_FOR;
        END_IF;
      END_FOR;
    END_IF;
  END_FOR;
END_FOR;

(* CHECK 3: TRANSPORTER_COLLISION *)
FOR vTi := 1 TO MAX_TRANSPORTERS DO
  FOR vQi := 1 TO ioTask[vTi].Count DO
    IF ioTask[vTi].Queue[vQi].Unit > 0 THEN
      vLIdx := ioTask[vTi].Queue[vQi].LiftStationTarget - MIN_STATION_INDEX;
      vSIdx := ioTask[vTi].Queue[vQi].SinkStationTarget - MIN_STATION_INDEX;
      IF vLIdx >= 1 AND vLIdx <= 30 THEN
        vLiftX := DINT_TO_REAL(Stations[ioTask[vTi].Queue[vQi].LiftStationTarget].XPosition);
  ELSE vLiftX := 0.0; END_IF;
      IF vSIdx >= 1 AND vSIdx <= 30 THEN
        vSinkX := DINT_TO_REAL(Stations[ioTask[vTi].Queue[vQi].SinkStationTarget].XPosition);
  ELSE vSinkX := 0.0; END_IF;
  IF vLiftX < vSinkX THEN vX1Min := vLiftX;
  vX1Max := vSinkX;
  ELSE vX1Min := vSinkX;
  vX1Max := vLiftX; END_IF;

      FOR vTj := vTi + 1 TO MAX_TRANSPORTERS DO
        FOR vQj := 1 TO ioTask[vTj].Count DO
          IF ioTask[vTj].Queue[vQj].Unit > 0 THEN
            vLIdx2 := ioTask[vTj].Queue[vQj].LiftStationTarget - MIN_STATION_INDEX;
            vSIdx2 := ioTask[vTj].Queue[vQj].SinkStationTarget - MIN_STATION_INDEX;
            IF vLIdx2 >= 1 AND vLIdx2 <= 30 THEN
              vLiftX2 := DINT_TO_REAL(Stations[ioTask[vTj].Queue[vQj].LiftStationTarget].XPosition);
  ELSE vLiftX2 := 0.0; END_IF;
            IF vSIdx2 >= 1 AND vSIdx2 <= 30 THEN
              vSinkX2 := DINT_TO_REAL(Stations[ioTask[vTj].Queue[vQj].SinkStationTarget].XPosition);
  ELSE vSinkX2 := 0.0; END_IF;
  IF vLiftX2 < vSinkX2 THEN vX2Min := vLiftX2;
  vX2Max := vSinkX2;
  ELSE vX2Min := vSinkX2;
  vX2Max := vLiftX2; END_IF;

  vXoStart := vX1Min; IF vX2Min > vXoStart THEN vXoStart := vX2Min; END_IF;
  vXoEnd := vX1Max; IF vX2Max < vXoEnd THEN vXoEnd := vX2Max; END_IF;

            IF vXoStart < vXoEnd THEN
              vToStart := ioTask[vTi].Queue[vQi].StartTime;
  IF ioTask[vTj].Queue[vQj].StartTime > vToStart THEN vToStart := ioTask[vTj].Queue[vQj].StartTime; END_IF;
              vToEnd := ioTask[vTi].Queue[vQi].FinishTime;
  IF ioTask[vTj].Queue[vQj].FinishTime < vToEnd THEN vToEnd := ioTask[vTj].Queue[vQj].FinishTime; END_IF;

              IF vToStart < vToEnd THEN
                vDeficitS := LINT_TO_REAL(vToEnd - vToStart) + 2.0;
  oHasConflict := TRUE;
  oConfType := 2;
                IF ioTask[vTi].Queue[vQi].StartTime <= ioTask[vTj].Queue[vQj].StartTime THEN
                  oConfUnit := ioTask[vTj].Queue[vQj].Unit;
                  oConfStage := ioTask[vTj].Queue[vQj].Stage;
                  oConfTrans := vTj;
                  oBlockedUnit := ioTask[vTi].Queue[vQi].Unit;
                  oBlockedStage := ioTask[vTi].Queue[vQi].Stage;
                ELSE
                  oConfUnit := ioTask[vTi].Queue[vQi].Unit;
                  oConfStage := ioTask[vTi].Queue[vQi].Stage;
                  oConfTrans := vTi;
                  oBlockedUnit := ioTask[vTj].Queue[vQj].Unit;
                  oBlockedStage := ioTask[vTj].Queue[vQj].Stage;
                END_IF;
  oDeficit := vDeficitS;
  oCheckedCount := vTotalTasks;
  TSK_FC_Analyze := TRUE; RETURN;
              END_IF;
            END_IF;
          END_IF;
        END_FOR;
      END_FOR;
    END_IF;
  END_FOR;
END_FOR;

oCheckedCount := vTotalTasks;

END_FUNCTION

(* ---- TSK_FC_NoTreatment.st ---- *)
(* ===========================================================================================
 *  TSK_FC_NoTreatment — Create no-treatment transfer tasks
 *
 *  Company : Galvatek part of the John Cockerill Group
 *  Author  : Jarmo Piipponen
 *  Created : 25.03.2026
 *
 * -------------------------------------------------------------------------------------------
 *  Scans units with a target and creates transfer tasks
 *  using the Ntt destination table.
 *
 *  VAR_IN_OUT: ioTask — only mutable array (inserts NTT tasks).
 *  All other globals are read-only via VAR_EXTERNAL.
 *
 *  ------------------------------------------------------------------------------------------
 *
 *  Changes:
 *
 *
 *
 *)

FUNCTION TSK_FC_NoTreatment : BOOL

(* Introduction of Variables ----------------------------------------------------------------*)

VAR_INPUT
  iTimeS                  : LINT;
END_VAR

VAR_IN_OUT  (* array sizes must match GVL_JC_Constants: 3=MAX_TRANSPORTERS *)
  ioTask                   : ARRAY[1..3] OF UDT_JC_TskQueueType;
END_VAR

VAR_EXTERNAL CONSTANT
    MAX_TRANSPORTERS        : INT;
    MAX_STATIONS_PER_STEP   : INT;
    MIN_STATION_INDEX        : INT;
    MAX_STATION_INDEX        : INT;
    MAX_UNITS               : INT;
    MAX_TASK_QUEUE          : INT;
    SCH_DISPATCH_MARGIN_S   : REAL;
    NOT_PROCESSED           : INT;
    PROCESSED               : INT;
    USED                    : INT;
END_VAR

VAR_EXTERNAL
  Unit                    : ARRAY[1..MAX_UNITS] OF UDT_JC_UnitType;
  Batch                   : ARRAY[1..MAX_UNITS] OF UDT_BatchType;
  Ntt                     : ARRAY[1..MAX_TRANSPORTERS] OF UDT_JC_NttTransporterType;
  TransporterStatus             : ARRAY[1..MAX_TRANSPORTERS] OF UDT_TransporterStatusType;
  Stations                 : ARRAY[MIN_STATION_INDEX..MAX_STATION_INDEX] OF UDT_StationType;
  StationOccupancy             : ARRAY[1..MAX_STATION_INDEX] OF UDT_JC_UnitAtStationType;
  Transporters                     : ARRAY[0..MAX_TRANSPORTERS] OF UDT_TransporterType;
  Move                    : ARRAY[1..MAX_TRANSPORTERS] OF UDT_JC_MoveTimesType;
END_VAR

VAR
  vUi                        : INT;
  vLoc                       : INT;
  vTgt                       : INT;
  vCovT                     : INT;
  vAi                        : INT;
  vCovers                    : BOOL;
  vDone                      : BOOL;
  vDest                      : UDT_JC_NttDestType;
  vNttIdx                   : INT;
  vOnPrimary                : BOOL;
  vOnFallback               : BOOL;
  vPrimaryFree              : BOOL;
  vDestStn                  : INT;
  vSi                        : INT;
  vStationIdx               : INT;
  vStnFree                  : BOOL;
  vUj                        : INT;
  vTi                        : INT;
  vAlready                   : BOOL;
  vQi2                       : INT;
  vXferS                    : REAL;
  vTaskStart                : LINT;
  vTaskEnd                  : LINT;
  vSlotStart                : LINT;
  vTmpMove                  : UDT_JC_MoveTimesType;
  vSlotEnd                  : LINT;
  vLatestEnd                : LINT;
  vTravelFromSink          : REAL;
  vTravelToLiftS          : REAL;
  vTransPos                 : INT;
  vNttDuration              : LINT;
  vSlotOk                   : BOOL;
  vSh                        : INT;

  (* Idle-stretch: extend blocking batch CalTime to make room for NTT -----------------------*)
  vStretchPending           : BOOL;
  vStretchUnitId           : INT;
  vStretchDeficit           : DINT;
  vStretchAvail             : DINT;

  (* Multi-transporter shared-area idle check -----------------------------------------------*)
  vOt                        : INT;
  vOq                        : INT;
  vOverlapConflict          : BOOL;
  vDestX                    : DINT;
  vAvoidDist                : DINT;
  vCovMinX                 : DINT;
  vCovMaxX                 : DINT;
  vOtMinX                  : DINT;
  vOtMaxX                  : DINT;
  vZoneMinX                : DINT;
  vZoneMaxX                : DINT;
  vDangerMin                : DINT;
  vDangerMax                : DINT;
  (* Shared-area timing: NTT split into own-area + shared-area portions ---------------------*)
  vLocIdx                   : INT;
  vLocX                     : DINT;
  vPhase2S                  : REAL;
  vSharedEntry              : LINT;
  vSharedTime               : REAL;
  vOtIdleOk                : BOOL;
  vOtIdleStart             : LINT;
  vOtIdleEnd               : LINT;
  vOtNextLift              : INT;
  vOtDispatchFrom          : INT;
  vOtTravelToNext         : REAL;

  (* Idle-stretch for other transporter: widen idle gap by extending blocker CalTime --------*)
  vOtStretchPending        : BOOL;
  vOtStretchUnitId        : INT;
  vOtStretchDeficit        : DINT;
  vOtStretchAvail          : DINT;
  vOtStretchNeed           : LINT;
  vOtStretchOk             : BOOL;
END_VAR

TSK_FC_NoTreatment := TRUE;

FOR vUi := 1 TO MAX_UNITS DO
  vTgt := Unit[vUi].Target;
  vLoc := Unit[vUi].location;

  IF vTgt >= 1 AND vTgt <= 5 AND vLoc >= MIN_STATION_INDEX THEN

    IF vTgt = 3 AND (Batch[vUi].BatchCode = 0 OR Batch[vUi].State <> NOT_PROCESSED) THEN
      CONTINUE;
    END_IF;

    vAlready := FALSE;
    FOR vTi := 1 TO MAX_TRANSPORTERS DO
      IF NOT vAlready THEN
        IF TransporterStatus[vTi].Phase > 0 AND StationOccupancy[vTi].UnitId = vUi THEN
          vAlready := TRUE;
        END_IF;
        FOR vQi2 := 1 TO ioTask[vTi].Count DO
          IF NOT vAlready THEN
            IF ioTask[vTi].Queue[vQi2].Unit = vUi THEN
              vAlready := TRUE;
            END_IF;
          END_IF;
        END_FOR;
      END_IF;
    END_FOR;

    IF NOT vAlready THEN

    vDone := FALSE;
    FOR vCovT := 1 TO MAX_TRANSPORTERS DO
      IF NOT vDone THEN

      vCovers := FALSE;
      FOR vAi := 1 TO 4 DO
        IF NOT vCovers THEN
          IF Transporters[vCovT].TaskArea[vAi].MinLift > 0 OR Transporters[vCovT].TaskArea[vAi].MaxLift > 0 THEN
            IF vLoc >= Transporters[vCovT].TaskArea[vAi].MinLift AND vLoc <= Transporters[vCovT].TaskArea[vAi].MaxLift THEN
              vCovers := TRUE;
            END_IF;
          END_IF;
        END_IF;
      END_FOR;

      IF vCovers AND TransporterStatus[vCovT].IsActive
         AND (TransporterStatus[vCovT].Phase = 0 OR vTgt = 5) THEN

        IF vTgt = 2 THEN
          IF Batch[vUi].BatchCode = 0 THEN vNttIdx := 6;
          ELSIF Batch[vUi].State = PROCESSED THEN vNttIdx := 8;
  ELSE vNttIdx := 7; END_IF;
        ELSIF vTgt = 3 THEN vNttIdx := 7;
  ELSE vNttIdx := vTgt; END_IF;

        vDest := Ntt[vCovT].Target[vNttIdx];

        vOnPrimary := FALSE;
        FOR vSi := 1 TO vDest.StationCount DO
  IF vDest.Stations[vSi] = vLoc THEN vOnPrimary := TRUE; END_IF;
        END_FOR;

        IF NOT vOnPrimary THEN

          vOnFallback := FALSE;
          FOR vSi := 1 TO vDest.FallbackCount DO
  IF vDest.FallbackStations[vSi] = vLoc THEN vOnFallback := TRUE; END_IF;
          END_FOR;

          vPrimaryFree := FALSE;
          FOR vSi := 1 TO vDest.StationCount DO
            vStationIdx := vDest.Stations[vSi];
            IF vStationIdx <> vLoc AND vStationIdx >= MIN_STATION_INDEX AND vStationIdx <= MAX_STATION_INDEX THEN
              vStnFree := TRUE;
              FOR vUj := 1 TO MAX_UNITS DO
  IF Unit[vUj].location = vStationIdx AND Unit[vUj].Status = USED THEN vStnFree := FALSE; END_IF;
              END_FOR;
  IF vStnFree THEN vPrimaryFree := TRUE; END_IF;
            END_IF;
          END_FOR;

          vDestStn := 0;

          IF vOnFallback AND NOT vPrimaryFree THEN
            vDestStn := 0;
          ELSIF vOnFallback AND vPrimaryFree THEN
            FOR vSi := 1 TO vDest.StationCount DO
              IF vDestStn = 0 THEN
                vStationIdx := vDest.Stations[vSi];
                IF vStationIdx <> vLoc AND vStationIdx >= MIN_STATION_INDEX AND vStationIdx <= MAX_STATION_INDEX THEN
                  vStnFree := TRUE;
                  FOR vUj := 1 TO MAX_UNITS DO
  IF Unit[vUj].location = vStationIdx AND Unit[vUj].Status = USED THEN vStnFree := FALSE; END_IF;
                  END_FOR;
  IF vStnFree THEN vDestStn := vStationIdx; END_IF;
                END_IF;
              END_IF;
            END_FOR;
          ELSE
            FOR vSi := 1 TO vDest.StationCount DO
              IF vDestStn = 0 THEN
                vStationIdx := vDest.Stations[vSi];
                IF vStationIdx <> vLoc AND vStationIdx >= MIN_STATION_INDEX AND vStationIdx <= MAX_STATION_INDEX THEN
                  vStnFree := TRUE;
                  FOR vUj := 1 TO MAX_UNITS DO
  IF Unit[vUj].location = vStationIdx AND Unit[vUj].Status = USED THEN vStnFree := FALSE; END_IF;
                  END_FOR;
  IF vStnFree THEN vDestStn := vStationIdx; END_IF;
                END_IF;
              END_IF;
            END_FOR;

            IF vDestStn = 0 THEN
              FOR vSi := 1 TO vDest.FallbackCount DO
                IF vDestStn = 0 THEN
                  vStationIdx := vDest.FallbackStations[vSi];
                  IF vStationIdx <> vLoc AND vStationIdx >= MIN_STATION_INDEX AND vStationIdx <= MAX_STATION_INDEX THEN
                    vStnFree := TRUE;
                    FOR vUj := 1 TO MAX_UNITS DO
  IF Unit[vUj].location = vStationIdx AND Unit[vUj].Status = USED THEN vStnFree := FALSE; END_IF;
                    END_FOR;
  IF vStnFree THEN vDestStn := vStationIdx; END_IF;
                  END_IF;
                END_IF;
              END_FOR;
            END_IF;
          END_IF;

          IF vDestStn > 0 THEN
            vTmpMove := Move[vCovT];
            vXferS := STC_FC_CalcTransferTime(
              iFromStn            := vLoc,
              iToStn              := vDestStn,
              iMove                := vTmpMove,
              iFromDroppingX10   := Stations[vLoc].DrippingTime,
              iToDeviceDelayX10 := Stations[vDestStn].DeviceDelay,
              iDripTrayDelayX10 := Transporters[vCovT].DripTrayDelay);

            (* ── Travel-to: time for transporter to reach lift station ── *)
            vTravelToLiftS := 0.0;
            IF TransporterStatus[vCovT].Phase = 0 THEN
              vTransPos := TransporterStatus[vCovT].CurrentStation;
            ELSE
              vTransPos := TransporterStatus[vCovT].SinkStationTarget;
            END_IF;
            IF vTransPos > 0 AND vTransPos <> vLoc THEN
              vTravelToLiftS := STC_FC_CalcHorizontalTravel(
                iFromStn := vTransPos,
                iToStn   := vLoc,
                iMove     := vTmpMove);
            END_IF;

            vTaskStart := iTimeS + REAL_TO_LINT(vTravelToLiftS);
            vTaskEnd   := vTaskStart + REAL_TO_LINT(vXferS);
            vNttDuration := vTaskEnd - vTaskStart;

            vSlotOk := FALSE;
            vStretchPending := FALSE;
            vOtStretchPending := FALSE;

            IF ioTask[vCovT].Count = 0 THEN
              vSlotOk := TRUE;
            ELSE
              IF ioTask[vCovT].Queue[1].StartTime > vTaskStart THEN
                vSlotStart := vTaskStart;
                vSlotEnd   := ioTask[vCovT].Queue[1].StartTime;
                vTravelFromSink := STC_FC_CalcHorizontalTravel(
                  iFromStn := vDestStn,
                  iToStn   := ioTask[vCovT].Queue[1].LiftStationTarget,
                  iMove     := Move[vCovT]);
                vLatestEnd := vSlotEnd - REAL_TO_LINT(vTravelFromSink) - 1;
                IF vTaskStart >= vSlotStart AND vTaskEnd <= vLatestEnd THEN
                  vSlotOk := TRUE;
                END_IF;

                (* ── Idle-stretch: NTT slightly too long for idle window ──
                   Check if the blocking batch's treatment CalTime can be
                   extended (up to MaxTime) to widen the idle gap.  Only flag
                   the intent here; the actual Batch write happens after
                   the multi-transporter overlap check passes. *)
                IF NOT vSlotOk AND vLatestEnd > 0 THEN
                  vStretchDeficit := LINT_TO_DINT(vTaskEnd - vLatestEnd);
                  IF vStretchDeficit > 0 THEN
                    vStretchUnitId := ioTask[vCovT].Queue[1].Unit;
                    IF vStretchUnitId >= 1 AND vStretchUnitId <= MAX_UNITS THEN
                      vStretchAvail := Batch[vStretchUnitId].MaxTime
                                     - Batch[vStretchUnitId].CalTime;
                      IF vStretchAvail >= vStretchDeficit THEN
                        vStretchPending := TRUE;
                        vSlotOk := TRUE;
                      END_IF;
                    END_IF;
                  END_IF;
                END_IF;
              END_IF;
            END_IF;

            IF NOT vSlotOk THEN
              IF ioTask[vCovT].Count > 0
                 AND ioTask[vCovT].Queue[1].SinkStationTarget = vLoc THEN
                vSlotOk := TRUE;
              ELSE
                vDestStn := 0;
              END_IF;
            END_IF;
          END_IF;

          (* ── Multi-transporter shared-area idle check ──
             If vDestStn is on the shared drive area between two transporters,
             the other transporter must have an idle window covering the time
             when THIS transporter is physically on the shared area.

             NTT transfer phases:
               Phase 2: lift + drip + tray  (nostin on vielä lift-asemalla)
               Phase 3: horizontal travel   (nostin liikkuu kohti vDest)
               Phase 4: lower + tray + dev  (nostin on vDest-asemalla)

             If lift station is NOT on shared area:
               vSharedEntry = vTaskStart + vPhase2S  (travel starts)
               vSharedTime  = vXferS - vPhase2S
             If lift station IS on shared area:
               vSharedEntry = vTaskStart  (vAlready there)
               vSharedTime  = vXferS
          *)
          IF vDestStn > 0 THEN
            vOverlapConflict := FALSE;
            vDestX := Stations[vDestStn].XPosition;
            vAvoidDist := Transporters[vCovT].AvoidanceWidth;
            vCovMinX := Transporters[vCovT].DrivePosMin;
            vCovMaxX := Transporters[vCovT].DrivePosMax;

            FOR vOt := 1 TO MAX_TRANSPORTERS DO
              IF vOt <> vCovT AND NOT vOverlapConflict
                 AND TransporterStatus[vOt].IsActive THEN
                vOtMinX := Transporters[vOt].DrivePosMin;
                vOtMaxX := Transporters[vOt].DrivePosMax;

                IF vCovMinX > vOtMinX THEN vZoneMinX := vCovMinX;
  ELSE vZoneMinX := vOtMinX; END_IF;
                IF vCovMaxX < vOtMaxX THEN vZoneMaxX := vCovMaxX;
  ELSE vZoneMaxX := vOtMaxX; END_IF;

                IF vZoneMinX >= vZoneMaxX THEN CONTINUE; END_IF;
                IF vDestX < vZoneMinX OR vDestX > vZoneMaxX THEN CONTINUE; END_IF;

                vDangerMin := vZoneMinX - vAvoidDist;
                vDangerMax := vZoneMaxX + vAvoidDist;

                (* ── Calculate shared-area entry time and duration ── *)
                vLocX := Stations[vLoc].XPosition;
                IF vLocX >= vDangerMin AND vLocX <= vDangerMax THEN
                  vSharedEntry := vTaskStart;
                  vSharedTime  := vXferS;
                ELSE
                  vLocIdx := vLoc - MIN_STATION_INDEX;
                  IF vLocIdx >= 1 AND vLocIdx <= 25 THEN
                    vPhase2S := INT_TO_REAL(Move[vCovT].LiftTime[vLocIdx]) / 10.0
                              + INT_TO_REAL(Stations[vLoc].DrippingTime) / 10.0
                              + INT_TO_REAL(Transporters[vCovT].DripTrayDelay) / 10.0;
                  ELSE
                    vPhase2S := 0.0;
                  END_IF;
                  vSharedEntry := vTaskStart + REAL_TO_LINT(vPhase2S);
                  vSharedTime  := vXferS - vPhase2S;
  IF vSharedTime < 1.0 THEN vSharedTime := 1.0; END_IF;
                END_IF;

                (* ── Check: does other transporter have an idle window
                     that starts ≤ vSharedEntry and lasts ≥ vSharedTime? ── *)
                vOtIdleOk := FALSE;

                IF ioTask[vOt].Count = 0 AND TransporterStatus[vOt].Phase = 0 THEN
                  vOtIdleOk := TRUE;
                ELSIF ioTask[vOt].Count = 0
                      AND TransporterStatus[vOt].Phase >= 1
                      AND TransporterStatus[vOt].Phase <= 4 THEN
                  (* Transporter executing task, nothing queued after.
                     Idle starts at current task finish. *)
                  vOtIdleStart := TransporterStatus[vOt].CurrentTaskFinishTime;
                  IF vOtIdleStart <= vSharedEntry THEN
                    vOtIdleOk := TRUE;
                  END_IF;
                ELSE
                  IF ioTask[vOt].Count > 0 THEN
                    IF TransporterStatus[vOt].Phase >= 1 AND TransporterStatus[vOt].Phase <= 4 THEN
                      (* Idle gap: current task finish → next queued start *)
                      vOtIdleStart := TransporterStatus[vOt].CurrentTaskFinishTime;
                      vOtDispatchFrom := TransporterStatus[vOt].SinkStationTarget;
                    ELSE
                      vOtIdleStart := vTaskStart;
                      vOtDispatchFrom := TransporterStatus[vOt].CurrentStation;
                    END_IF;
                    vOtNextLift := ioTask[vOt].Queue[1].LiftStationTarget;
                    vOtTravelToNext := 0.0;
                    IF vOtDispatchFrom > 0
                       AND vOtNextLift > 0
                       AND vOtDispatchFrom <> vOtNextLift THEN
                      vOtTravelToNext := STC_FC_CalcHorizontalTravel(
                        iFromStn := vOtDispatchFrom,
                        iToStn   := vOtNextLift,
                        iMove     := Move[vOt]);
                    END_IF;
                    vOtIdleEnd := ioTask[vOt].Queue[1].StartTime
                                 - REAL_TO_LINT(vOtTravelToNext)
                                 - REAL_TO_LINT(SCH_DISPATCH_MARGIN_S);
                    IF vOtIdleEnd < vOtIdleStart THEN
                      vOtIdleEnd := vOtIdleStart;
                    END_IF;
                    IF vOtIdleStart <= vSharedEntry
                       AND vOtIdleEnd >= vSharedEntry + REAL_TO_LINT(vSharedTime) THEN
                      vOtIdleOk := TRUE;
                    END_IF;
                  END_IF;

                  IF NOT vOtIdleOk THEN
                    FOR vOq := 1 TO ioTask[vOt].Count - 1 DO
                      IF NOT vOtIdleOk THEN
                        vOtIdleStart := ioTask[vOt].Queue[vOq].FinishTime;
                        vOtDispatchFrom := ioTask[vOt].Queue[vOq].SinkStationTarget;
                        vOtNextLift := ioTask[vOt].Queue[vOq + 1].LiftStationTarget;
                        vOtTravelToNext := 0.0;
                        IF vOtDispatchFrom > 0
                           AND vOtNextLift > 0
                           AND vOtDispatchFrom <> vOtNextLift THEN
                          vOtTravelToNext := STC_FC_CalcHorizontalTravel(
                            iFromStn := vOtDispatchFrom,
                            iToStn   := vOtNextLift,
                            iMove     := Move[vOt]);
                        END_IF;
                        vOtIdleEnd := ioTask[vOt].Queue[vOq + 1].StartTime
                                     - REAL_TO_LINT(vOtTravelToNext)
                                     - REAL_TO_LINT(SCH_DISPATCH_MARGIN_S);
                        IF vOtIdleEnd < vOtIdleStart THEN
                          vOtIdleEnd := vOtIdleStart;
                        END_IF;
                        IF vOtIdleStart <= vSharedEntry
                           AND vOtIdleEnd >= vSharedEntry + REAL_TO_LINT(vSharedTime) THEN
                          vOtIdleOk := TRUE;
                        END_IF;
                      END_IF;
                    END_FOR;
                  END_IF;

                  IF NOT vOtIdleOk AND ioTask[vOt].Count > 0 THEN
                    vOtIdleStart := ioTask[vOt].Queue[ioTask[vOt].Count].FinishTime;
                    IF vOtIdleStart <= vSharedEntry THEN
                      vOtIdleOk := TRUE;
                    END_IF;
                  END_IF;
                END_IF;

                IF NOT vOtIdleOk THEN
                  (* ── Idle-stretch for other transporter ──
                     Try to widen the nearest idle gap by extending the
                     blocking batch CalTime (up to MaxTime).  Only tasks
                     with Stage > 0 (regular, not NTT) are candidates. *)
                  vOtStretchOk := FALSE;

                  (* Try gap before first task *)
                  IF ioTask[vOt].Count > 0
                     AND ioTask[vOt].Queue[1].Stage > 0 THEN
                    IF TransporterStatus[vOt].Phase >= 1 AND TransporterStatus[vOt].Phase <= 4 THEN
                      vOtIdleStart := TransporterStatus[vOt].CurrentTaskFinishTime;
                      vOtDispatchFrom := TransporterStatus[vOt].SinkStationTarget;
                    ELSE
                      vOtIdleStart := vTaskStart;
                      vOtDispatchFrom := TransporterStatus[vOt].CurrentStation;
                    END_IF;
                    vOtNextLift := ioTask[vOt].Queue[1].LiftStationTarget;
                    vOtTravelToNext := 0.0;
                    IF vOtDispatchFrom > 0
                       AND vOtNextLift > 0
                       AND vOtDispatchFrom <> vOtNextLift THEN
                      vOtTravelToNext := STC_FC_CalcHorizontalTravel(
                        iFromStn := vOtDispatchFrom,
                        iToStn   := vOtNextLift,
                        iMove     := Move[vOt]);
                    END_IF;
                    vOtIdleEnd := ioTask[vOt].Queue[1].StartTime
                                 - REAL_TO_LINT(vOtTravelToNext)
                                 - REAL_TO_LINT(SCH_DISPATCH_MARGIN_S);
                    IF vOtIdleEnd < vOtIdleStart THEN
                      vOtIdleEnd := vOtIdleStart;
                    END_IF;

                    IF vOtIdleStart <= vSharedEntry
                       AND vOtIdleEnd > vSharedEntry THEN
                      vOtStretchNeed := vSharedEntry
                                       + REAL_TO_LINT(vSharedTime)
                                       - vOtIdleEnd;
                      IF vOtStretchNeed > LINT#0 THEN
                        vOtStretchUnitId := ioTask[vOt].Queue[1].Unit;
                        IF vOtStretchUnitId >= 1
                           AND vOtStretchUnitId <= MAX_UNITS THEN
                          vOtStretchAvail :=
                            Batch[vOtStretchUnitId].MaxTime
                          - Batch[vOtStretchUnitId].CalTime;
                          IF vOtStretchAvail >= LINT_TO_DINT(vOtStretchNeed) THEN
                            vOtStretchDeficit := LINT_TO_DINT(vOtStretchNeed);
                            vOtStretchPending := TRUE;
                            vOtStretchOk      := TRUE;
                          END_IF;
                        END_IF;
                      END_IF;
                    END_IF;
                  END_IF;

                  (* Try gaps between tasks *)
                  IF NOT vOtStretchOk THEN
                    FOR vOq := 1 TO ioTask[vOt].Count - 1 DO
                      IF NOT vOtStretchOk
                         AND ioTask[vOt].Queue[vOq + 1].Stage > 0 THEN
                        vOtIdleStart := ioTask[vOt].Queue[vOq].FinishTime;
                        vOtDispatchFrom := ioTask[vOt].Queue[vOq].SinkStationTarget;
                        vOtNextLift := ioTask[vOt].Queue[vOq + 1].LiftStationTarget;
                        vOtTravelToNext := 0.0;
                        IF vOtDispatchFrom > 0
                           AND vOtNextLift > 0
                           AND vOtDispatchFrom <> vOtNextLift THEN
                          vOtTravelToNext := STC_FC_CalcHorizontalTravel(
                            iFromStn := vOtDispatchFrom,
                            iToStn   := vOtNextLift,
                            iMove     := Move[vOt]);
                        END_IF;
                        vOtIdleEnd := ioTask[vOt].Queue[vOq + 1].StartTime
                                     - REAL_TO_LINT(vOtTravelToNext)
                                     - REAL_TO_LINT(SCH_DISPATCH_MARGIN_S);
                        IF vOtIdleEnd < vOtIdleStart THEN
                          vOtIdleEnd := vOtIdleStart;
                        END_IF;

                        IF vOtIdleStart <= vSharedEntry
                           AND vOtIdleEnd > vSharedEntry THEN
                          vOtStretchNeed := vSharedEntry
                                           + REAL_TO_LINT(vSharedTime)
                                           - vOtIdleEnd;
                          IF vOtStretchNeed > LINT#0 THEN
                            vOtStretchUnitId := ioTask[vOt].Queue[vOq + 1].Unit;
                            IF vOtStretchUnitId >= 1
                               AND vOtStretchUnitId <= MAX_UNITS THEN
                              vOtStretchAvail :=
                                Batch[vOtStretchUnitId].MaxTime
                              - Batch[vOtStretchUnitId].CalTime;
                              IF vOtStretchAvail >= LINT_TO_DINT(vOtStretchNeed) THEN
                                vOtStretchDeficit := LINT_TO_DINT(vOtStretchNeed);
                                vOtStretchPending := TRUE;
                                vOtStretchOk      := TRUE;
                              END_IF;
                            END_IF;
                          END_IF;
                        END_IF;
                      END_IF;
                    END_FOR;
                  END_IF;

                  IF vOtStretchOk THEN
                    vOtIdleOk := TRUE;
                  ELSE
                    vOverlapConflict := TRUE;
                  END_IF;
                END_IF;
              END_IF;
            END_FOR;

  IF vOverlapConflict THEN vDestStn := 0; END_IF;
          END_IF;

          IF vDestStn > 0 THEN
            (* ── Commit idle-stretch: extend blocking batch CalTime ── *)
            IF vStretchPending THEN
              Batch[vStretchUnitId].CalTime :=
                Batch[vStretchUnitId].CalTime + vStretchDeficit;
              vStretchPending := FALSE;
            END_IF;

            (* ── Commit other-transporter idle-stretch ── *)
            IF vOtStretchPending THEN
              Batch[vOtStretchUnitId].CalTime :=
                Batch[vOtStretchUnitId].CalTime + vOtStretchDeficit;
              vOtStretchPending := FALSE;
            END_IF;

            IF ioTask[vCovT].Count < MAX_TASK_QUEUE THEN
              FOR vSh := ioTask[vCovT].Count TO 1 BY -1 DO
                ioTask[vCovT].Queue[vSh + 1] := ioTask[vCovT].Queue[vSh];
              END_FOR;
              ioTask[vCovT].Queue[1].Unit         := vUi;
              ioTask[vCovT].Queue[1].Stage        := 0;
              ioTask[vCovT].Queue[1].LiftStationTarget := vLoc;
              ioTask[vCovT].Queue[1].SinkStationTarget := vDestStn;
              ioTask[vCovT].Queue[1].StartTime   := vTaskStart;
              ioTask[vCovT].Queue[1].FinishTime  := vTaskEnd;
              ioTask[vCovT].Queue[1].CalcTime    := 0;
              ioTask[vCovT].Queue[1].MinTime     := 0;
              ioTask[vCovT].Queue[1].MaxTime     := 0;
              ioTask[vCovT].Queue[1].NttPrimary := 0;
              FOR vSi := 1 TO vDest.StationCount DO
                IF vDest.Stations[vSi] = vDestStn THEN
                  ioTask[vCovT].Queue[1].NttPrimary := 1;
                END_IF;
              END_FOR;
              ioTask[vCovT].Count := ioTask[vCovT].Count + 1;
              vDone := TRUE;
            END_IF;
          END_IF;

        END_IF; (* NOT vOnPrimary *)
      END_IF; (* vCovers + idle *)
      END_IF; (* NOT vDone *)
    END_FOR; (* transporter loop *)
    END_IF; (* NOT vAlready *)
  END_IF; (* valid target *)
END_FOR;

END_FUNCTION

(* ---- TSK_FC_Resolve.st ---- *)
(* ===========================================================================================
 *  TSK_FC_Resolve — Conflict resolution
 *
 *  Company : Galvatek part of the John Cockerill Group
 *  Author  : Jarmo Piipponen
 *  Created : 25.03.2026
 *
 * -------------------------------------------------------------------------------------------
 *  Four sequential resolution phases:
 *  1. ADVANCE (chain bottleneck + suffix flex_down)
 *  2. DELAY (single-stage flex_up)
 *  3. PRECEDING_DELAY (conf stage-1)
 *  4. DELAY_PREV_PAST_NEXT (force order swap)
 *
 *  VAR_IN_OUT: ioSchedule, ioTask, ioBatch, ioLocks,
 *  ioLockCnt — caller passes live or workspace arrays.
 *
 *  ------------------------------------------------------------------------------------------
 *
 *  Changes:
 *
 *
 *
 *)

FUNCTION TSK_FC_Resolve : BOOL

(* Introduction of Variables ----------------------------------------------------------------*)

VAR_INPUT
  iConfUnit               : INT;
  iConfStage              : INT;
  iConfTrans              : INT;
  iBlockedUnit            : INT;
  iBlockedStage           : INT;
  iDeficit                 : REAL;
END_VAR

VAR_IN_OUT  (* array sizes must match GVL_JC_Constants: 50=MAX_LOCKS, 10=MAX_UNITS, 3=MAX_TRANSPORTERS *)
  ioLocks                  : ARRAY[1..50] OF UDT_JC_TskLockType;
  ioLockCnt               : INT;
  ioSchedule               : ARRAY[1..10] OF UDT_JC_TskScheduleType;
  ioTask                   : ARRAY[1..3] OF UDT_JC_TskQueueType;
  ioBatch                  : ARRAY[1..10] OF UDT_BatchType;
END_VAR

VAR_EXTERNAL CONSTANT
    MAX_TRANSPORTERS        : INT;
    MAX_UNITS               : INT;
    SCH_TSK_FLEX_FACTOR     : REAL;
END_VAR

VAR_OUTPUT
  oSolved                  : BOOL;
  oTotalDelay             : REAL;
  oTotalAdv               : REAL;
END_VAR

VAR
  vRemain                    : REAL;
  vCap                       : REAL;
  vAmount                    : REAL;
  vStageFlex                : REAL;
  vIsLockedAdv             : BOOL;
  vIsLockedDel             : BOOL;
  vCanAdvance               : BOOL;
  vCanDelay                 : BOOL;
  vLockI                    : INT;
  vPrevConfStage           : INT;
  vIsPcsLocked             : BOOL;
  vPrevSinkStn             : INT;
  vNextLiftStn             : INT;
  vIsBlkAdvLocked         : BOOL;
  vQi                        : INT;
  vChainFlex                : REAL;
  vSuffixFlex               : REAL;
  vEarlierStg               : INT;
  vEarlierFlex              : REAL;
  vChainAmount              : REAL;
  vSuffixAmount             : REAL;
  vSchedBlocked             : INT;
  vSchedConf                : INT;
  vSchedPrevConf           : INT;
  vTmpSi                    : INT;
  vCapRemain                : REAL;
END_VAR

TSK_FC_Resolve := FALSE;
oSolved      := FALSE;
oTotalDelay := 0.0;
oTotalAdv   := 0.0;
vRemain        := iDeficit;

IF vRemain <= 0.1 THEN
  oSolved := TRUE;
  TSK_FC_Resolve := TRUE;
  RETURN;
END_IF;

(* Lock check: blocked stage locked DELAY? cannot ADVANCE *)
vIsLockedAdv := FALSE;
FOR vLockI := 1 TO ioLockCnt DO
  IF ioLocks[vLockI].Unit = iBlockedUnit
     AND ioLocks[vLockI].Stage = iBlockedStage
     AND ioLocks[vLockI].Direction = 2 THEN
    vIsLockedAdv := TRUE;
  END_IF;
END_FOR;

(* Lock check: conf stage locked ADVANCE? cannot DELAY *)
vIsLockedDel := FALSE;
FOR vLockI := 1 TO ioLockCnt DO
  IF ioLocks[vLockI].Unit = iConfUnit
     AND ioLocks[vLockI].Stage = iConfStage
     AND ioLocks[vLockI].Direction = 1 THEN
    vIsLockedDel := TRUE;
  END_IF;
END_FOR;

vCanAdvance := NOT vIsLockedAdv;
vCanDelay   := NOT vIsLockedDel;

(* Map ProgramStage to schedule array index *)
vSchedBlocked := 0;
IF iBlockedUnit >= 1 AND iBlockedUnit <= MAX_UNITS THEN
  FOR vTmpSi := 1 TO ioSchedule[iBlockedUnit].StageCount DO
    IF ioSchedule[iBlockedUnit].Stages[vTmpSi].ProgramStage = iBlockedStage THEN
      vSchedBlocked := vTmpSi; EXIT;
    END_IF;
  END_FOR;
END_IF;

vSchedConf := 0;
IF iConfUnit >= 1 AND iConfUnit <= MAX_UNITS THEN
  FOR vTmpSi := 1 TO ioSchedule[iConfUnit].StageCount DO
    IF ioSchedule[iConfUnit].Stages[vTmpSi].ProgramStage = iConfStage THEN
      vSchedConf := vTmpSi; EXIT;
    END_IF;
  END_FOR;
END_IF;

(* ================================================================ *)
(* PHASE 1: ADVANCE -- advance blocked batch                       *)
(* ================================================================ *)
IF vCanAdvance
   AND iBlockedUnit >= 1 AND iBlockedUnit <= MAX_UNITS
   AND iBlockedStage >= 1 THEN
IF vSchedBlocked >= 1 AND vSchedBlocked <= ioSchedule[iBlockedUnit].StageCount THEN

  (* Absolute flex vCap: use (MaxTime - MinTime) range, not (CalcTime - MinTime).
     This prevents cumulative drift when CalcTime is adjusted across rounds. *)
  vStageFlex := DINT_TO_REAL(
    ioSchedule[iBlockedUnit].Stages[vSchedBlocked].MaxTime
    - ioSchedule[iBlockedUnit].Stages[vSchedBlocked].MinTime);
  IF vStageFlex < 0.0 THEN vStageFlex := 0.0; END_IF;
  vStageFlex := vStageFlex * SCH_TSK_FLEX_FACTOR;
  (* Cap to actual remaining advance room *)
  vCapRemain := DINT_TO_REAL(
    ioSchedule[iBlockedUnit].Stages[vSchedBlocked].CalcTime
    - ioSchedule[iBlockedUnit].Stages[vSchedBlocked].MinTime);
  IF vCapRemain < 0.0 THEN vCapRemain := 0.0; END_IF;
  IF vStageFlex > vCapRemain THEN vStageFlex := vCapRemain; END_IF;

  IF vStageFlex > 0.1 THEN
    IF ioBatch[iBlockedUnit].CurStage = iBlockedStage THEN vCap := 0.9;
  ELSE vCap := 0.5; END_IF;

    (* Chain bottleneck search *)
    vChainFlex := vStageFlex;
    FOR vEarlierStg := 1 TO vSchedBlocked - 1 DO
      vEarlierFlex := DINT_TO_REAL(
        ioSchedule[iBlockedUnit].Stages[vEarlierStg].CalcTime
        - ioSchedule[iBlockedUnit].Stages[vEarlierStg].MinTime);
  IF vEarlierFlex < 0.0 THEN vEarlierFlex := 0.0; END_IF;
      IF vEarlierFlex > 0.0 AND vEarlierFlex < vChainFlex THEN
        vChainFlex := vEarlierFlex;
      END_IF;
    END_FOR;

    (* CHAIN_ADVANCE *)
    vChainAmount := vChainFlex * vCap;
  IF vChainAmount > vRemain THEN vChainAmount := vRemain; END_IF;

    IF vChainAmount > 0.1 THEN
      ioSchedule[iBlockedUnit].Stages[vSchedBlocked].CalcTime :=
        ioSchedule[iBlockedUnit].Stages[vSchedBlocked].CalcTime - REAL_TO_DINT(vChainAmount);
      ioSchedule[iBlockedUnit].Stages[vSchedBlocked].ExitTime :=
        ioSchedule[iBlockedUnit].Stages[vSchedBlocked].ExitTime - REAL_TO_LINT(vChainAmount);

      STC_FC_ShiftSchedule(iUnit := iBlockedUnit, iFromStage := iBlockedStage + 1,
                         iAmount := -vChainAmount, ioSchedule := ioSchedule, ioTask := ioTask);

      ioBatch[iBlockedUnit].CalTime :=
        ioBatch[iBlockedUnit].CalTime - REAL_TO_DINT(vChainAmount);
      IF ioBatch[iBlockedUnit].CalTime < ioBatch[iBlockedUnit].MinTime THEN
        ioBatch[iBlockedUnit].CalTime := ioBatch[iBlockedUnit].MinTime;
      END_IF;

      vRemain := vRemain - vChainAmount;
      oTotalAdv := oTotalAdv + vChainAmount;
    END_IF;

    (* SUFFIX_ADVANCE *)
    vSuffixFlex := vStageFlex - vChainFlex;
    IF vSuffixFlex > 0.1 AND vRemain > 0.1 THEN
      vSuffixAmount := vSuffixFlex * vCap;
  IF vSuffixAmount > vRemain THEN vSuffixAmount := vRemain; END_IF;

      IF vSuffixAmount > 0.1 THEN
        ioSchedule[iBlockedUnit].Stages[vSchedBlocked].CalcTime :=
          ioSchedule[iBlockedUnit].Stages[vSchedBlocked].CalcTime - REAL_TO_DINT(vSuffixAmount);
        ioSchedule[iBlockedUnit].Stages[vSchedBlocked].ExitTime :=
          ioSchedule[iBlockedUnit].Stages[vSchedBlocked].ExitTime - REAL_TO_LINT(vSuffixAmount);

        STC_FC_ShiftSchedule(iUnit := iBlockedUnit, iFromStage := iBlockedStage + 1,
                           iAmount := -vSuffixAmount, ioSchedule := ioSchedule, ioTask := ioTask);

        ioBatch[iBlockedUnit].CalTime :=
          ioBatch[iBlockedUnit].CalTime - REAL_TO_DINT(vSuffixAmount);
        IF ioBatch[iBlockedUnit].CalTime < ioBatch[iBlockedUnit].MinTime THEN
          ioBatch[iBlockedUnit].CalTime := ioBatch[iBlockedUnit].MinTime;
        END_IF;

        vRemain := vRemain - vSuffixAmount;
        oTotalAdv := oTotalAdv + vSuffixAmount;
      END_IF;
    END_IF;

    (* Record lock: ADVANCE on blocked stage *)
    IF ioLockCnt < 50 THEN
      ioLockCnt := ioLockCnt + 1;
      ioLocks[ioLockCnt].Unit := iBlockedUnit;
      ioLocks[ioLockCnt].Stage := iBlockedStage;
      ioLocks[ioLockCnt].Direction := 1;
    END_IF;

    IF vRemain <= 0.1 THEN
  oSolved := TRUE;
  TSK_FC_Resolve := TRUE; RETURN;
    END_IF;
  END_IF;
END_IF;
END_IF;

(* ================================================================ *)
(* PHASE 2: DELAY -- delay conflict batch                          *)
(* ================================================================ *)
IF vCanDelay AND vRemain > 0.1
   AND iConfUnit >= 1 AND iConfUnit <= MAX_UNITS
   AND iConfStage >= 1 THEN
IF vSchedConf >= 1 AND vSchedConf <= ioSchedule[iConfUnit].StageCount THEN

  (* Absolute flex vCap: use (MaxTime - MinTime) range, not (MaxTime - CalcTime).
     This prevents cumulative drift when CalcTime is adjusted across rounds. *)
  vStageFlex := DINT_TO_REAL(
    ioSchedule[iConfUnit].Stages[vSchedConf].MaxTime
    - ioSchedule[iConfUnit].Stages[vSchedConf].MinTime);
  IF vStageFlex < 0.0 THEN vStageFlex := 0.0; END_IF;
  vStageFlex := vStageFlex * SCH_TSK_FLEX_FACTOR;
  (* Cap to actual remaining delay room *)
  vCapRemain := DINT_TO_REAL(
    ioSchedule[iConfUnit].Stages[vSchedConf].MaxTime
    - ioSchedule[iConfUnit].Stages[vSchedConf].CalcTime);
  IF vCapRemain < 0.0 THEN vCapRemain := 0.0; END_IF;
  IF vStageFlex > vCapRemain THEN vStageFlex := vCapRemain; END_IF;

  IF vStageFlex > 0.1 THEN
    IF ioBatch[iConfUnit].CurStage = iConfStage THEN vCap := 0.9;
  ELSE vCap := 0.5; END_IF;
    vAmount := vStageFlex * vCap;
  IF vAmount > vRemain THEN vAmount := vRemain; END_IF;

    ioSchedule[iConfUnit].Stages[vSchedConf].CalcTime :=
      ioSchedule[iConfUnit].Stages[vSchedConf].CalcTime + REAL_TO_DINT(vAmount);
    ioSchedule[iConfUnit].Stages[vSchedConf].ExitTime :=
      ioSchedule[iConfUnit].Stages[vSchedConf].ExitTime + REAL_TO_LINT(vAmount);

    STC_FC_ShiftSchedule(iUnit := iConfUnit, iFromStage := iConfStage + 1,
                       iAmount := vAmount, ioSchedule := ioSchedule, ioTask := ioTask);

    IF ioBatch[iConfUnit].CurStage = iConfStage THEN
      ioBatch[iConfUnit].CalTime :=
        ioBatch[iConfUnit].CalTime + REAL_TO_DINT(vAmount);
      IF ioBatch[iConfUnit].CalTime > ioBatch[iConfUnit].MaxTime THEN
        ioBatch[iConfUnit].CalTime := ioBatch[iConfUnit].MaxTime;
      END_IF;
    END_IF;

    vRemain := vRemain - vAmount;
    oTotalDelay := oTotalDelay + vAmount;

    IF ioLockCnt < 50 THEN
      ioLockCnt := ioLockCnt + 1;
      ioLocks[ioLockCnt].Unit := iConfUnit;
      ioLocks[ioLockCnt].Stage := iConfStage;
      ioLocks[ioLockCnt].Direction := 2;
    END_IF;

    IF vRemain <= 0.1 THEN
  oSolved := TRUE;
  TSK_FC_Resolve := TRUE; RETURN;
    END_IF;
  END_IF;
END_IF;
END_IF;

(* ================================================================ *)
(* PHASE 3: PRECEDING_DELAY -- delay conf batch at stage-1         *)
(* ================================================================ *)
vPrevConfStage := iConfStage - 1;

vSchedPrevConf := 0;
IF iConfUnit >= 1 AND iConfUnit <= MAX_UNITS AND vPrevConfStage >= 1 THEN
  FOR vTmpSi := 1 TO ioSchedule[iConfUnit].StageCount DO
    IF ioSchedule[iConfUnit].Stages[vTmpSi].ProgramStage = vPrevConfStage THEN
  vSchedPrevConf := vTmpSi; EXIT;
    END_IF;
  END_FOR;
END_IF;

IF vRemain > 0.1 AND vPrevConfStage >= 1 AND iConfUnit >= 1 AND iConfUnit <= MAX_UNITS
   AND vSchedPrevConf >= 1 THEN
  vIsPcsLocked := FALSE;
  FOR vLockI := 1 TO ioLockCnt DO
    IF ioLocks[vLockI].Unit = iConfUnit
       AND ioLocks[vLockI].Stage = vPrevConfStage
       AND ioLocks[vLockI].Direction = 1 THEN
      vIsPcsLocked := TRUE;
    END_IF;
  END_FOR;

  IF NOT vIsPcsLocked THEN
    (* Flex vCap: min + factor × (max - min); available room = flex_cap - CalcTime *)
    vStageFlex := DINT_TO_REAL(
      ioSchedule[iConfUnit].Stages[vSchedPrevConf].MinTime
      + REAL_TO_DINT(SCH_TSK_FLEX_FACTOR * DINT_TO_REAL(
          ioSchedule[iConfUnit].Stages[vSchedPrevConf].MaxTime
        - ioSchedule[iConfUnit].Stages[vSchedPrevConf].MinTime))
      - ioSchedule[iConfUnit].Stages[vSchedPrevConf].CalcTime);
  IF vStageFlex < 0.0 THEN vStageFlex := 0.0; END_IF;

    IF vStageFlex > 0.1 THEN
      IF ioBatch[iConfUnit].CurStage = vPrevConfStage THEN vCap := 0.9;
  ELSE vCap := 0.5; END_IF;
      vAmount := vStageFlex * vCap;
  IF vAmount > vRemain THEN vAmount := vRemain; END_IF;

      ioSchedule[iConfUnit].Stages[vSchedPrevConf].CalcTime :=
        ioSchedule[iConfUnit].Stages[vSchedPrevConf].CalcTime + REAL_TO_DINT(vAmount);
      ioSchedule[iConfUnit].Stages[vSchedPrevConf].ExitTime :=
        ioSchedule[iConfUnit].Stages[vSchedPrevConf].ExitTime + REAL_TO_LINT(vAmount);
      STC_FC_ShiftSchedule(iUnit := iConfUnit, iFromStage := vPrevConfStage + 1,
                         iAmount := vAmount, ioSchedule := ioSchedule, ioTask := ioTask);

      IF ioBatch[iConfUnit].CurStage = iConfStage THEN
        ioBatch[iConfUnit].CalTime :=
          ioBatch[iConfUnit].CalTime + REAL_TO_DINT(vAmount);
        IF ioBatch[iConfUnit].CalTime > ioBatch[iConfUnit].MaxTime THEN
          ioBatch[iConfUnit].CalTime := ioBatch[iConfUnit].MaxTime;
        END_IF;
      END_IF;

      vRemain := vRemain - vAmount;
      oTotalDelay := oTotalDelay + vAmount;

      IF ioLockCnt < 50 THEN
        ioLockCnt := ioLockCnt + 1;
        ioLocks[ioLockCnt].Unit := iConfUnit;
        ioLocks[ioLockCnt].Stage := vPrevConfStage;
        ioLocks[ioLockCnt].Direction := 2;
      END_IF;

      IF vRemain <= 0.1 THEN
  oSolved := TRUE;
  TSK_FC_Resolve := TRUE; RETURN;
      END_IF;
    END_IF;
  END_IF;
END_IF;

(* ================================================================ *)
(* PHASE 4: DELAY_PREV_PAST_NEXT -- force order swap               *)
(* ================================================================ *)
IF vRemain > 0.1 AND iBlockedUnit >= 1 AND iBlockedUnit <= MAX_UNITS THEN
  vPrevSinkStn := 0;
  vNextLiftStn := 0;
  IF iConfTrans >= 1 AND iConfTrans <= MAX_TRANSPORTERS THEN
    FOR vQi := 1 TO ioTask[iConfTrans].Count DO
      IF ioTask[iConfTrans].Queue[vQi].Unit = iBlockedUnit
         AND ioTask[iConfTrans].Queue[vQi].Stage = iBlockedStage THEN
        vPrevSinkStn := ioTask[iConfTrans].Queue[vQi].SinkStationTarget;
      END_IF;
      IF ioTask[iConfTrans].Queue[vQi].Unit = iConfUnit
         AND ioTask[iConfTrans].Queue[vQi].Stage = iConfStage THEN
        vNextLiftStn := ioTask[iConfTrans].Queue[vQi].LiftStationTarget;
      END_IF;
    END_FOR;
  END_IF;

  IF NOT (vPrevSinkStn > 0 AND vNextLiftStn > 0 AND vPrevSinkStn = vNextLiftStn) THEN
    vIsBlkAdvLocked := FALSE;
    FOR vLockI := 1 TO ioLockCnt DO
      IF ioLocks[vLockI].Unit = iBlockedUnit
         AND ioLocks[vLockI].Stage = iBlockedStage
         AND ioLocks[vLockI].Direction = 1 THEN
        vIsBlkAdvLocked := TRUE;
      END_IF;
    END_FOR;

    IF NOT vIsBlkAdvLocked THEN
      (* Flex vCap: min + factor × (max - min); available room = flex_cap - CalcTime *)
      vStageFlex := DINT_TO_REAL(
        ioSchedule[iBlockedUnit].Stages[vSchedBlocked].MinTime
        + REAL_TO_DINT(SCH_TSK_FLEX_FACTOR * DINT_TO_REAL(
            ioSchedule[iBlockedUnit].Stages[vSchedBlocked].MaxTime
          - ioSchedule[iBlockedUnit].Stages[vSchedBlocked].MinTime))
        - ioSchedule[iBlockedUnit].Stages[vSchedBlocked].CalcTime);
  IF vStageFlex < 0.0 THEN vStageFlex := 0.0; END_IF;

      IF vStageFlex > 0.1 THEN
        IF ioBatch[iBlockedUnit].CurStage = iBlockedStage THEN vCap := 0.9;
  ELSE vCap := 0.5; END_IF;
        vAmount := vStageFlex * vCap;
  IF vAmount > vRemain THEN vAmount := vRemain; END_IF;

        ioSchedule[iBlockedUnit].Stages[vSchedBlocked].CalcTime :=
          ioSchedule[iBlockedUnit].Stages[vSchedBlocked].CalcTime + REAL_TO_DINT(vAmount);
        ioSchedule[iBlockedUnit].Stages[vSchedBlocked].ExitTime :=
          ioSchedule[iBlockedUnit].Stages[vSchedBlocked].ExitTime + REAL_TO_LINT(vAmount);
        STC_FC_ShiftSchedule(iUnit := iBlockedUnit, iFromStage := iBlockedStage + 1,
                           iAmount := vAmount, ioSchedule := ioSchedule, ioTask := ioTask);

        IF ioBatch[iBlockedUnit].CurStage = iBlockedStage THEN
          ioBatch[iBlockedUnit].CalTime :=
            ioBatch[iBlockedUnit].CalTime + REAL_TO_DINT(vAmount);
          IF ioBatch[iBlockedUnit].CalTime > ioBatch[iBlockedUnit].MaxTime THEN
            ioBatch[iBlockedUnit].CalTime := ioBatch[iBlockedUnit].MaxTime;
          END_IF;
        END_IF;

        vRemain := vRemain - vAmount;
        oTotalDelay := oTotalDelay + vAmount;

        IF ioLockCnt < 50 THEN
          ioLockCnt := ioLockCnt + 1;
          ioLocks[ioLockCnt].Unit := iBlockedUnit;
          ioLocks[ioLockCnt].Stage := iBlockedStage;
          ioLocks[ioLockCnt].Direction := 2;
        END_IF;

        IF vRemain <= 0.1 THEN
  oSolved := TRUE;
  TSK_FC_Resolve := TRUE; RETURN;
        END_IF;
      END_IF;
    END_IF;
  END_IF;
END_IF;

END_FUNCTION
